LIN {X 0,Y 248.743,Z 466.9,A -85,B 0,C 180,E1 -20308.54,E2 -20308.54} C_VEL
LIN {X 0,Y 247.758,Z 471.99,A -85,B 0,C 180,E1 -20311.566,E2 -20311.566} C_VEL
LIN {X 0,Y 246.638,Z 476.028,A -85,B 0,C 180,E1 -20313.789,E2 -20313.789} C_VEL
LIN {X 0,Y 245.403,Z 479.129,A -85,B 0,C 180,E1 -20315.464,E2 -20315.464} C_VEL
LIN {X 0,Y 244.484,Z 480.76,A -85,B 0,C 180,E1 -20316.269,E2 -20316.269} C_VEL
LIN {X 0,Y 239.749,Z 485.852,A -85,B 0,C 180,E1 -20318.505,E2 -20318.505} C_VEL
LIN {X 0,Y 235.404,Z 489.582,A -85,B 0,C 180,E1 -20320.828,E2 -20320.828} C_VEL
LIN {X 0,Y 232.82,Z 491.419,A -85,B 0,C 180,E1 -20322.43,E2 -20322.43} C_VEL
LIN {X 0,Y 230.431,Z 492.703,A -85,B 0,C 180,E1 -20324.068,E2 -20324.068} C_VEL
LIN {X 0,Y 228.241,Z 493.449,A -85,B 0,C 180,E1 -20325.739,E2 -20325.739} C_VEL
LIN {X 0,Y 226.236,Z 493.719,A -85,B 0,C 180,E1 -20327.441,E2 -20327.441} C_VEL
LIN {X 0,Y 224.375,Z 493.441,A -85,B 0,C 180,E1 -20329.168,E2 -20329.168} C_VEL
LIN {X 0,Y 222.889,Z 492.598,A -85,B 0,C 180,E1 -20330.929,E2 -20330.929} C_VEL
LIN {X 0,Y 221.691,Z 491.23,A -85,B 0,C 180,E1 -20332.715,E2 -20332.715} C_VEL
LIN {X 0,Y 220.302,Z 488.075,A -85,B 0,C 180,E1 -20335.426,E2 -20335.426} C_VEL
LIN {X 0,Y 219.514,Z 483.587,A -85,B 0,C 180,E1 -20338.165,E2 -20338.165} C_VEL
LIN {X 0,Y 219.226,Z 477.6,A -85,B 0,C 180,E1 -20340.919,E2 -20340.919} C_VEL
LIN {X 0,Y 219.359,Z 471.25,A -85,B 0,C 180,E1 -20343.214,E2 -20343.214} C_VEL
LIN {X 0,Y 219.828,Z 463.432,A -85,B 0,C 180,E1 -20345.504,E2 -20345.504} C_VEL
LIN {X 0,Y 220.117,Z 454.301,A -85,B 0,C 180,E1 -20347.658,E2 -20347.658} C_VEL
LIN {X 0,Y 220.624,Z 443.788,A -85,B 0,C 180,E1 -20349.628,E2 -20349.628} C_VEL
LIN {X 0,Y 221.055,Z 434.685,A -85,B 0,C 180,E1 -20350.997,E2 -20350.997} C_VEL
LIN {X 0,Y 219.764,Z 422.117,A -85,B 0,C 180,E1 -20352.466,E2 -20352.466} C_VEL
LIN {X 0,Y 219.404,Z 416.978,A -85,B 0,C 180,E1 -20352.958,E2 -20352.958} C_VEL
LIN {X 0,Y 219.691,Z 410.88,A -85,B 0,C 180,E1 -20357.693,E2 -20357.693} C_VEL
LIN {X 0,Y 220.166,Z 404.789,A -85,B 0,C 180,E1 -20362.523,E2 -20362.523} C_VEL
LIN {X 0,Y 220.698,Z 399.342,A -85,B 0,C 180,E1 -20366.919,E2 -20366.919} C_VEL
LIN {X 0,Y 221.276,Z 394.44,A -85,B 0,C 180,E1 -20370.956,E2 -20370.956} C_VEL
LIN {X 0,Y 221.123,Z 392.931,A -85,B 0,C 180,E1 -20372.443,E2 -20372.443} C_VEL
LIN {X 0,Y 220.841,Z 392.976,A -85,B 0,C 180,E1 -20377.288,E2 -20377.288} C_VEL
LIN {X 0,Y 220.773,Z 392.981,A -85,B 0,C 180,E1 -20381.952,E2 -20381.952} C_VEL
LIN {X 0,Y 220.778,Z 392.982,A -85,B 0,C 180,E1 -20385.547,E2 -20385.547} C_VEL
LIN {X 0,Y 220.809,Z 392.979,A -85,B 0,C 180,E1 -20390.463,E2 -20390.463} C_VEL
LIN {X 0,Y 220.803,Z 392.98,A -85,B 0,C 180,E1 -20395.045,E2 -20395.045} C_VEL
LIN {X 0,Y 220.871,Z 392.968,A -85,B 0,C 180,E1 -20399.395,E2 -20399.395} C_VEL
LIN {X 0,Y 220.898,Z 392.967,A -85,B 0,C 180,E1 -20403.55,E2 -20403.55} C_VEL
LIN {X 0,Y 220.882,Z 392.967,A -85,B 0,C 180,E1 -20407.554,E2 -20407.554} C_VEL
LIN {X 0,Y 220.988,Z 392.958,A -85,B 0,C 180,E1 -20412.571,E2 -20412.571} C_VEL
LIN {X 0,Y 221.015,Z 392.949,A -85,B 0,C 180,E1 -20417.139,E2 -20417.139} C_VEL
LIN {X 0,Y 221.208,Z 392.929,A -85,B 0,C 180,E1 -20420.859,E2 -20420.859} C_VEL
LIN {X 0,Y 221.263,Z 392.922,A -85,B 0,C 180,E1 -20422.701,E2 -20422.701} C_VEL
LIN {X 0,Y 221.515,Z 392.893,A -85,B 0,C 180,E1 -20428.182,E2 -20428.182} C_VEL
LIN {X 0,Y 221.516,Z 392.893,A -85,B 0,C 180,E1 -20431.818,E2 -20431.818} C_VEL
LIN {X 0,Y 221.292,Z 392.918,A -85,B 0,C 180,E1 -20437.298,E2 -20437.298} C_VEL
LIN {X 0,Y 221.115,Z 392.939,A -85,B 0,C 180,E1 -20440.994,E2 -20440.994} C_VEL
LIN {X 0,Y 221.02,Z 392.952,A -85,B 0,C 180,E1 -20446.629,E2 -20446.629} C_VEL
LIN {X 0,Y 220.913,Z 392.963,A -85,B 0,C 180,E1 -20450.484,E2 -20450.484} C_VEL
LIN {X 0,Y 220.875,Z 392.97,A -85,B 0,C 180,E1 -20454.434,E2 -20454.434} C_VEL
LIN {X 0,Y 220.838,Z 392.973,A -85,B 0,C 180,E1 -20458.513,E2 -20458.513} C_VEL
LIN {X 0,Y 220.827,Z 392.976,A -85,B 0,C 180,E1 -20462.754,E2 -20462.754} C_VEL
LIN {X 0,Y 220.84,Z 392.976,A -85,B 0,C 180,E1 -20467.288,E2 -20467.288} C_VEL
LIN {X 0,Y 220.773,Z 392.983,A -85,B 0,C 180,E1 -20471.952,E2 -20471.952} C_VEL
LIN {X 0,Y 220.769,Z 392.983,A -85,B 0,C 180,E1 -20475.544,E2 -20475.544} C_VEL
LIN {X 0,Y 220.808,Z 392.978,A -85,B 0,C 180,E1 -20480.463,E2 -20480.463} C_VEL
LIN {X 0,Y 220.802,Z 392.979,A -85,B 0,C 180,E1 -20485.045,E2 -20485.045} C_VEL
LIN {X 0,Y 220.87,Z 392.972,A -85,B 0,C 180,E1 -20489.395,E2 -20489.395} C_VEL
LIN {X 0,Y 220.897,Z 392.965,A -85,B 0,C 180,E1 -20493.549,E2 -20493.549} C_VEL
LIN {X 0,Y 220.88,Z 392.97,A -85,B 0,C 180,E1 -20497.553,E2 -20497.553} C_VEL
LIN {X 0,Y 220.986,Z 392.956,A -85,B 0,C 180,E1 -20502.571,E2 -20502.571} C_VEL
LIN {X 0,Y 221.029,Z 392.952,A -85,B 0,C 180,E1 -20507.139,E2 -20507.139} C_VEL
LIN {X 0,Y 221.26,Z 392.921,A -85,B 0,C 180,E1 -20510.862,E2 -20510.862} C_VEL
LIN {X 0,Y 221.313,Z 392.917,A -85,B 0,C 180,E1 -20512.702,E2 -20512.702} C_VEL
LIN {X 0,Y 221.515,Z 392.891,A -85,B 0,C 180,E1 -20518.182,E2 -20518.182} C_VEL
LIN {X 0,Y 221.517,Z 392.889,A -85,B 0,C 180,E1 -20521.818,E2 -20521.818} C_VEL
LIN {X 0,Y 221.313,Z 392.913,A -85,B 0,C 180,E1 -20527.298,E2 -20527.298} C_VEL
LIN {X 0,Y 221.119,Z 392.94,A -85,B 0,C 180,E1 -20530.994,E2 -20530.994} C_VEL
LIN {X 0,Y 221.018,Z 392.95,A -85,B 0,C 180,E1 -20536.63,E2 -20536.63} C_VEL
LIN {X 0,Y 220.894,Z 392.969,A -85,B 0,C 180,E1 -20540.486,E2 -20540.486} C_VEL
LIN {X 0,Y 220.869,Z 392.97,A -85,B 0,C 180,E1 -20544.435,E2 -20544.435} C_VEL
LIN {X 0,Y 220.828,Z 392.977,A -85,B 0,C 180,E1 -20548.515,E2 -20548.515} C_VEL
LIN {X 0,Y 220.824,Z 392.975,A -85,B 0,C 180,E1 -20552.755,E2 -20552.755} C_VEL
LIN {X 0,Y 220.839,Z 392.975,A -85,B 0,C 180,E1 -20557.288,E2 -20557.288} C_VEL
LIN {X 0,Y 220.777,Z 392.981,A -85,B 0,C 180,E1 -20561.951,E2 -20561.951} C_VEL
LIN {X 0,Y 220.889,Z 392.973,A -85,B 0,C 180,E1 -20565.812,E2 -20565.812} C_VEL
LIN {X 0,Y 222.459,Z 401.177,A -85,B 0,C 180,E1 -20570.814,E2 -20570.814} C_VEL
LIN {X 0,Y 223.883,Z 407.84,A -85,B 0,C 180,E1 -20574.704,E2 -20574.704} C_VEL
LIN {X 0,Y 225.236,Z 413.607,A -85,B 0,C 180,E1 -20577.964,E2 -20577.964} C_VEL
LIN {X 0,Y 225.146,Z 415.498,A -85,B 0,C 180,E1 -20578.999,E2 -20578.999} C_VEL
LIN {X 0,Y 222.346,Z 426.144,A -85,B 0,C 180,E1 -20584.741,E2 -20584.741} C_VEL
LIN {X 0,Y 220.633,Z 436.118,A -85,B 0,C 180,E1 -20590.218,E2 -20590.218} C_VEL
LIN {X 0,Y 220.815,Z 450.1,A -85,B 0,C 180,E1 -20591.321,E2 -20591.321} C_VEL
LIN {X 0,Y 221.565,Z 462.255,A -85,B 0,C 180,E1 -20592.619,E2 -20592.619} C_VEL
LIN {X 0,Y 221.177,Z 467.503,A -85,B 0,C 180,E1 -20593.309,E2 -20593.309} C_VEL
LIN {X 0,Y 219.653,Z 472.431,A -85,B 0,C 180,E1 -20594.084,E2 -20594.084} C_VEL
LIN {X 0,Y 215.142,Z 483.065,A -85,B 0,C 180,E1 -20596.213,E2 -20596.213} C_VEL
LIN {X 0,Y 214.264,Z 487.568,A -85,B 0,C 180,E1 -20597.255,E2 -20597.255} C_VEL
LIN {X 0,Y 213.864,Z 496.597,A -85,B 0,C 180,E1 -20599.588,E2 -20599.588} C_VEL
LIN {X 0,Y 213.658,Z 503.978,A -85,B 0,C 180,E1 -20601.94,E2 -20601.94} C_VEL
LIN {X 0,Y 213.802,Z 510.152,A -85,B 0,C 180,E1 -20604.341,E2 -20604.341} C_VEL
LIN {X 0,Y 213.841,Z 515.818,A -85,B 0,C 180,E1 -20607.174,E2 -20607.174} C_VEL
LIN {X 0,Y 213.76,Z 518.769,A -85,B 0,C 180,E1 -20609.058,E2 -20609.058} C_VEL
LIN {X 0,Y 213.37,Z 522.06,A -85,B 0,C 180,E1 -20611.888,E2 -20611.888} C_VEL
LIN {X 0,Y 212.82,Z 523.57,A -85,B 0,C 180,E1 -20613.787,E2 -20613.787} C_VEL
LIN {X 0,Y 212.266,Z 525.354,A -85,B 0,C 180,E1 -20617.611,E2 -20617.611} C_VEL
LIN {X 0,Y 212.516,Z 525.684,A -85,B 0,C 180,E1 -20621.445,E2 -20621.445} C_VEL
LIN {X 0,Y 213.939,Z 524.599,A -85,B 0,C 180,E1 -20625.237,E2 -20625.237} C_VEL
LIN {X 0,Y 216.51,Z 522.127,A -85,B 0,C 180,E1 -20628.942,E2 -20628.942} C_VEL
LIN {X 0,Y 220.264,Z 518.23,A -85,B 0,C 180,E1 -20632.513,E2 -20632.513} C_VEL
LIN {X 0,Y 223.867,Z 514.286,A -85,B 0,C 180,E1 -20635.076,E2 -20635.076} C_VEL
LIN {X 0,Y 229.577,Z 507.575,A -85,B 0,C 180,E1 -20638.327,E2 -20638.327} C_VEL
LIN {X 0,Y 234.674,Z 501.249,A -85,B 0,C 180,E1 -20640.605,E2 -20640.605} C_VEL
LIN {X 0,Y 239.782,Z 493.834,A -85,B 0,C 180,E1 -20642.836,E2 -20642.836} C_VEL
LIN {X 0,Y 243.085,Z 487.19,A -85,B 0,C 180,E1 -20644.821,E2 -20644.821} C_VEL
LIN {X 0,Y 246.585,Z 477.943,A -85,B 0,C 180,E1 -20647.627,E2 -20647.627} C_VEL
LIN {X 0,Y 247.275,Z 475.617,A -85,B 0,C 180,E1 -20648.373,E2 -20648.373} C_VEL
LIN {X 0,Y 247.04,Z 473.044,A -85,B 0,C 180,E1 -20649.815,E2 -20649.815} C_VEL
LIN {X 0,Y 246.243,Z 470.086,A -85,B 0,C 180,E1 -20652.092,E2 -20652.092} C_VEL
LIN {X 0,Y 245.716,Z 467.717,A -85,B 0,C 180,E1 -20654.352,E2 -20654.352} C_VEL
LIN {X 0,Y 245.265,Z 466.253,A -85,B 0,C 180,E1 -20656.551,E2 -20656.551} C_VEL
LIN {X 0,Y 244.953,Z 465.624,A -85,B 0,C 180,E1 -20658.708,E2 -20658.708} C_VEL
LIN {X 0,Y 244.685,Z 465.81,A -85,B 0,C 180,E1 -20660.852,E2 -20660.852} C_VEL
LIN {X 0,Y 244.47,Z 466.992,A -85,B 0,C 180,E1 -20663.605,E2 -20663.605} C_VEL
LIN {X 0,Y 244.352,Z 467.904,A -85,B 0,C 180,E1 -20664.884,E2 -20664.884} C_VEL
LIN {X 0,Y 244.034,Z 469.82,A -85,B 0,C 180,E1 -20666.826,E2 -20666.826} C_VEL
LIN {X 0,Y 243.396,Z 472.34,A -85,B 0,C 180,E1 -20668.685,E2 -20668.685} C_VEL
LIN {X 0,Y 242.066,Z 476.535,A -85,B 0,C 180,E1 -20671.432,E2 -20671.432} C_VEL
LIN {X 0,Y 240.286,Z 480.703,A -85,B 0,C 180,E1 -20673.977,E2 -20673.977} C_VEL
LIN {X 0,Y 239.559,Z 482.111,A -85,B 0,C 180,E1 -20674.825,E2 -20674.825} C_VEL
LIN {X 0,Y 238.383,Z 483.655,A -85,B 0,C 180,E1 -20675.622,E2 -20675.622} C_VEL
LIN {X 0,Y 233.427,Z 488.207,A -85,B 0,C 180,E1 -20677.892,E2 -20677.892} C_VEL
LIN {X 0,Y 228.932,Z 491.524,A -85,B 0,C 180,E1 -20680.264,E2 -20680.264} C_VEL
LIN {X 0,Y 226.222,Z 493.059,A -85,B 0,C 180,E1 -20681.901,E2 -20681.901} C_VEL
LIN {X 0,Y 223.744,Z 494.077,A -85,B 0,C 180,E1 -20683.579,E2 -20683.579} C_VEL
LIN {X 0,Y 221.453,Z 494.605,A -85,B 0,C 180,E1 -20685.292,E2 -20685.292} C_VEL
LIN {X 0,Y 219.356,Z 494.613,A -85,B 0,C 180,E1 -20687.04,E2 -20687.04} C_VEL
LIN {X 0,Y 217.444,Z 494.086,A -85,B 0,C 180,E1 -20688.818,E2 -20688.818} C_VEL
LIN {X 0,Y 215.906,Z 493.026,A -85,B 0,C 180,E1 -20690.633,E2 -20690.633} C_VEL
LIN {X 0,Y 214.127,Z 490.391,A -85,B 0,C 180,E1 -20693.404,E2 -20693.404} C_VEL
LIN {X 0,Y 212.882,Z 486.483,A -85,B 0,C 180,E1 -20696.214,E2 -20696.214} C_VEL
LIN {X 0,Y 212.297,Z 481.155,A -85,B 0,C 180,E1 -20699.052,E2 -20699.052} C_VEL
LIN {X 0,Y 212.165,Z 474.239,A -85,B 0,C 180,E1 -20701.898,E2 -20701.898} C_VEL
LIN {X 0,Y 212.495,Z 466.979,A -85,B 0,C 180,E1 -20704.268,E2 -20704.268} C_VEL
LIN {X 0,Y 212.873,Z 459.912,A -85,B 0,C 180,E1 -20706.16,E2 -20706.16} C_VEL
LIN {X 0,Y 213.245,Z 450.42,A -85,B 0,C 180,E1 -20708.251,E2 -20708.251} C_VEL
LIN {X 0,Y 213.741,Z 439.494,A -85,B 0,C 180,E1 -20710.18,E2 -20710.18} C_VEL
LIN {X 0,Y 213.97,Z 434.77,A -85,B 0,C 180,E1 -20710.887,E2 -20710.887} C_VEL
LIN {X 0,Y 212.789,Z 423.368,A -85,B 0,C 180,E1 -20712.276,E2 -20712.276} C_VEL
LIN {X 0,Y 212.331,Z 417.259,A -85,B 0,C 180,E1 -20712.91,E2 -20712.91} C_VEL
LIN {X 0,Y 212.669,Z 410.519,A -85,B 0,C 180,E1 -20718.297,E2 -20718.297} C_VEL
LIN {X 0,Y 213.197,Z 404.385,A -85,B 0,C 180,E1 -20723.302,E2 -20723.302} C_VEL
LIN {X 0,Y 213.882,Z 398.208,A -85,B 0,C 180,E1 -20728.455,E2 -20728.455} C_VEL
LIN {X 0,Y 214.245,Z 394.452,A -85,B 0,C 180,E1 -20731.659,E2 -20731.659} C_VEL
LIN {X 0,Y 214.104,Z 393.807,A -85,B 0,C 180,E1 -20732.236,E2 -20732.236} C_VEL
LIN {X 0,Y 213.754,Z 393.857,A -85,B 0,C 180,E1 -20737.898,E2 -20737.898} C_VEL
LIN {X 0,Y 213.715,Z 393.861,A -85,B 0,C 180,E1 -20741.125,E2 -20741.125} C_VEL
LIN {X 0,Y 213.71,Z 393.86,A -85,B 0,C 180,E1 -20743.678,E2 -20743.678} C_VEL
LIN {X 0,Y 213.71,Z 393.864,A -85,B 0,C 180,E1 -20746.343,E2 -20746.343} C_VEL
LIN {X 0,Y 213.72,Z 393.861,A -85,B 0,C 180,E1 -20749.143,E2 -20749.143} C_VEL
LIN {X 0,Y 213.746,Z 393.857,A -85,B 0,C 180,E1 -20753.712,E2 -20753.712} C_VEL
LIN {X 0,Y 213.77,Z 393.856,A -85,B 0,C 180,E1 -20758.263,E2 -20758.263} C_VEL
LIN {X 0,Y 213.829,Z 393.85,A -85,B 0,C 180,E1 -20762.603,E2 -20762.603} C_VEL
LIN {X 0,Y 213.855,Z 393.843,A -85,B 0,C 180,E1 -20766.953,E2 -20766.953} C_VEL
LIN {X 0,Y 213.936,Z 393.838,A -85,B 0,C 180,E1 -20772.305,E2 -20772.305} C_VEL
LIN {X 0,Y 213.956,Z 393.829,A -85,B 0,C 180,E1 -20776.707,E2 -20776.707} C_VEL
LIN {X 0,Y 214.145,Z 393.81,A -85,B 0,C 180,E1 -20780.555,E2 -20780.555} C_VEL
LIN {X 0,Y 214.104,Z 393.813,A -85,B 0,C 180,E1 -20784.348,E2 -20784.348} C_VEL
LIN {X 0,Y 214.449,Z 393.773,A -85,B 0,C 180,E1 -20788.122,E2 -20788.122} C_VEL
LIN {X 0,Y 214.553,Z 393.761,A -85,B 0,C 180,E1 -20790,E2 -20790} C_VEL
LIN {X 0,Y 214.45,Z 393.773,A -85,B 0,C 180,E1 -20791.878,E2 -20791.878} C_VEL
LIN {X 0,Y 214.23,Z 393.799,A -85,B 0,C 180,E1 -20797.54,E2 -20797.54} C_VEL
LIN {X 0,Y 214.048,Z 393.821,A -85,B 0,C 180,E1 -20801.362,E2 -20801.362} C_VEL
LIN {X 0,Y 213.937,Z 393.834,A -85,B 0,C 180,E1 -20805.237,E2 -20805.237} C_VEL
LIN {X 0,Y 213.879,Z 393.842,A -85,B 0,C 180,E1 -20809.184,E2 -20809.184} C_VEL
LIN {X 0,Y 213.858,Z 393.843,A -85,B 0,C 180,E1 -20813.226,E2 -20813.226} C_VEL
LIN {X 0,Y 213.831,Z 393.85,A -85,B 0,C 180,E1 -20817.45,E2 -20817.45} C_VEL
LIN {X 0,Y 213.782,Z 393.855,A -85,B 0,C 180,E1 -20821.735,E2 -20821.735} C_VEL
LIN {X 0,Y 213.755,Z 393.856,A -85,B 0,C 180,E1 -20826.286,E2 -20826.286} C_VEL
LIN {X 0,Y 213.716,Z 393.863,A -85,B 0,C 180,E1 -20831.124,E2 -20831.124} C_VEL
LIN {X 0,Y 213.704,Z 393.864,A -85,B 0,C 180,E1 -20833.679,E2 -20833.679} C_VEL
LIN {X 0,Y 213.704,Z 393.861,A -85,B 0,C 180,E1 -20836.345,E2 -20836.345} C_VEL
LIN {X 0,Y 213.718,Z 393.863,A -85,B 0,C 180,E1 -20839.143,E2 -20839.143} C_VEL
LIN {X 0,Y 213.745,Z 393.857,A -85,B 0,C 180,E1 -20843.712,E2 -20843.712} C_VEL
LIN {X 0,Y 213.797,Z 393.853,A -85,B 0,C 180,E1 -20848.725,E2 -20848.725} C_VEL
LIN {X 0,Y 213.827,Z 393.849,A -85,B 0,C 180,E1 -20852.603,E2 -20852.603} C_VEL
LIN {X 0,Y 213.854,Z 393.848,A -85,B 0,C 180,E1 -20856.953,E2 -20856.953} C_VEL
LIN {X 0,Y 213.934,Z 393.833,A -85,B 0,C 180,E1 -20862.305,E2 -20862.305} C_VEL
LIN {X 0,Y 213.983,Z 393.832,A -85,B 0,C 180,E1 -20866.708,E2 -20866.708} C_VEL
LIN {X 0,Y 214.199,Z 393.802,A -85,B 0,C 180,E1 -20870.558,E2 -20870.558} C_VEL
LIN {X 0,Y 214.25,Z 393.794,A -85,B 0,C 180,E1 -20872.46,E2 -20872.46} C_VEL
LIN {X 0,Y 214.448,Z 393.771,A -85,B 0,C 180,E1 -20878.122,E2 -20878.122} C_VEL
LIN {X 0,Y 214.553,Z 393.755,A -85,B 0,C 180,E1 -20880,E2 -20880} C_VEL
LIN {X 0,Y 214.45,Z 393.769,A -85,B 0,C 180,E1 -20881.878,E2 -20881.878} C_VEL
LIN {X 0,Y 214.25,Z 393.793,A -85,B 0,C 180,E1 -20887.539,E2 -20887.539} C_VEL
LIN {X 0,Y 214.049,Z 393.82,A -85,B 0,C 180,E1 -20891.362,E2 -20891.362} C_VEL
LIN {X 0,Y 213.935,Z 393.833,A -85,B 0,C 180,E1 -20895.237,E2 -20895.237} C_VEL
LIN {X 0,Y 213.841,Z 393.845,A -85,B 0,C 180,E1 -20899.187,E2 -20899.187} C_VEL
LIN {X 0,Y 213.849,Z 393.845,A -85,B 0,C 180,E1 -20903.227,E2 -20903.227} C_VEL
LIN {X 0,Y 213.83,Z 393.846,A -85,B 0,C 180,E1 -20907.45,E2 -20907.45} C_VEL
LIN {X 0,Y 213.771,Z 393.857,A -85,B 0,C 180,E1 -20911.737,E2 -20911.737} C_VEL
LIN {X 0,Y 213.754,Z 393.858,A -85,B 0,C 180,E1 -20916.286,E2 -20916.286} C_VEL
LIN {X 0,Y 213.718,Z 393.861,A -85,B 0,C 180,E1 -20921.124,E2 -20921.124} C_VEL
LIN {X 0,Y 213.845,Z 393.927,A -85,B 0,C 180,E1 -20925.628,E2 -20925.628} C_VEL
LIN {X 0,Y 215.277,Z 401.464,A -85,B 0,C 180,E1 -20930.397,E2 -20930.397} C_VEL
LIN {X 0,Y 216.886,Z 408.878,A -85,B 0,C 180,E1 -20934.888,E2 -20934.888} C_VEL
LIN {X 0,Y 218.154,Z 414.264,A -85,B 0,C 180,E1 -20938.047,E2 -20938.047} C_VEL
LIN {X 0,Y 218.011,Z 415.857,A -85,B 0,C 180,E1 -20938.95,E2 -20938.95} C_VEL
LIN {X 0,Y 215.155,Z 426.4,A -85,B 0,C 180,E1 -20944.872,E2 -20944.872} C_VEL
LIN {X 0,Y 213.561,Z 435.845,A -85,B 0,C 180,E1 -20950.287,E2 -20950.287} C_VEL
LIN {X 0,Y 213.676,Z 448.936,A -85,B 0,C 180,E1 -20951.344,E2 -20951.344} C_VEL
LIN {X 0,Y 214.525,Z 462.513,A -85,B 0,C 180,E1 -20952.852,E2 -20952.852} C_VEL
LIN {X 0,Y 215.247,Z 471.51,A -85,B 0,C 180,E1 -20954.13,E2 -20954.13} C_VEL
LIN {X 0,Y 214.623,Z 481.89,A -85,B 0,C 180,E1 -20956.025,E2 -20956.025} C_VEL
LIN {X 0,Y 214.264,Z 487.568,A -85,B 0,C 180,E1 -20957.255,E2 -20957.255} C_VEL
LIN {X 0,Y 213.411,Z 491.817,A -85,B 0,C 180,E1 -20958.335,E2 -20958.335} C_VEL
LIN {X 0,Y 210.34,Z 497.938,A -85,B 0,C 180,E1 -20960.277,E2 -20960.277} C_VEL
LIN {X 0,Y 207.438,Z 503.473,A -85,B 0,C 180,E1 -20962.415,E2 -20962.415} C_VEL
LIN {X 0,Y 206.869,Z 506.757,A -85,B 0,C 180,E1 -20963.78,E2 -20963.78} C_VEL
LIN {X 0,Y 206.918,Z 511.845,A -85,B 0,C 180,E1 -20966.105,E2 -20966.105} C_VEL
LIN {X 0,Y 206.926,Z 516.83,A -85,B 0,C 180,E1 -20969.027,E2 -20969.027} C_VEL
LIN {X 0,Y 206.469,Z 520.34,A -85,B 0,C 180,E1 -20971.951,E2 -20971.951} C_VEL
LIN {X 0,Y 205.508,Z 523.233,A -85,B 0,C 180,E1 -20975.889,E2 -20975.889} C_VEL
LIN {X 0,Y 205.324,Z 524.57,A -85,B 0,C 180,E1 -20979.855,E2 -20979.855} C_VEL
LIN {X 0,Y 206.105,Z 524.49,A -85,B 0,C 180,E1 -20983.81,E2 -20983.81} C_VEL
LIN {X 0,Y 208.268,Z 523.06,A -85,B 0,C 180,E1 -20987.68,E2 -20987.68} C_VEL
LIN {X 0,Y 211.572,Z 520.267,A -85,B 0,C 180,E1 -20991.432,E2 -20991.432} C_VEL
LIN {X 0,Y 216.125,Z 516.029,A -85,B 0,C 180,E1 -20995.008,E2 -20995.008} C_VEL
LIN {X 0,Y 221.832,Z 510.272,A -85,B 0,C 180,E1 -20998.374,E2 -20998.374} C_VEL
LIN {X 0,Y 228.7,Z 502.714,A -85,B 0,C 180,E1 -21001.495,E2 -21001.495} C_VEL
LIN {X 0,Y 234.074,Z 495.802,A -85,B 0,C 180,E1 -21003.743,E2 -21003.743} C_VEL
LIN {X 0,Y 237.657,Z 489.653,A -85,B 0,C 180,E1 -21005.736,E2 -21005.736} C_VEL
LIN {X 0,Y 241.689,Z 480.782,A -85,B 0,C 180,E1 -21008.645,E2 -21008.645} C_VEL
LIN {X 0,Y 242.148,Z 479.508,A -85,B 0,C 180,E1 -21009.118,E2 -21009.118} C_VEL
LIN {X 0,Y 241.82,Z 476.811,A -85,B 0,C 180,E1 -21010.919,E2 -21010.919} C_VEL
LIN {X 0,Y 241.097,Z 473.14,A -85,B 0,C 180,E1 -21014.395,E2 -21014.395} C_VEL
LIN {X 0,Y 240.662,Z 471.59,A -85,B 0,C 180,E1 -21016.893,E2 -21016.893} C_VEL
LIN {X 0,Y 240.138,Z 471.113,A -85,B 0,C 180,E1 -21019.92,E2 -21019.92} C_VEL
LIN {X 0,Y 239.779,Z 471.659,A -85,B 0,C 180,E1 -21022.315,E2 -21022.315} C_VEL
LIN {X 0,Y 239.515,Z 472.537,A -85,B 0,C 180,E1 -21024.066,E2 -21024.066} C_VEL
LIN {X 0,Y 239.055,Z 474.137,A -85,B 0,C 180,E1 -21026.042,E2 -21026.042} C_VEL
LIN {X 0,Y 238.25,Z 476.24,A -85,B 0,C 180,E1 -21027.929,E2 -21027.929} C_VEL
LIN {X 0,Y 236.606,Z 479.884,A -85,B 0,C 180,E1 -21030.653,E2 -21030.653} C_VEL
LIN {X 0,Y 234.5,Z 483.698,A -85,B 0,C 180,E1 -21033.285,E2 -21033.285} C_VEL
LIN {X 0,Y 233.681,Z 484.944,A -85,B 0,C 180,E1 -21034.145,E2 -21034.145} C_VEL
LIN {X 0,Y 232.279,Z 486.419,A -85,B 0,C 180,E1 -21034.938,E2 -21034.938} C_VEL
LIN {X 0,Y 227.131,Z 490.472,A -85,B 0,C 180,E1 -21037.246,E2 -21037.246} C_VEL
LIN {X 0,Y 222.456,Z 493.355,A -85,B 0,C 180,E1 -21039.664,E2 -21039.664} C_VEL
LIN {X 0,Y 219.631,Z 494.616,A -85,B 0,C 180,E1 -21041.338,E2 -21041.338} C_VEL
LIN {X 0,Y 217.044,Z 495.367,A -85,B 0,C 180,E1 -21043.057,E2 -21043.057} C_VEL
LIN {X 0,Y 214.674,Z 495.645,A -85,B 0,C 180,E1 -21044.817,E2 -21044.817} C_VEL
LIN {X 0,Y 212.475,Z 495.394,A -85,B 0,C 180,E1 -21046.612,E2 -21046.612} C_VEL
LIN {X 0,Y 210.524,Z 494.633,A -85,B 0,C 180,E1 -21048.446,E2 -21048.446} C_VEL
LIN {X 0,Y 208.931,Z 493.335,A -85,B 0,C 180,E1 -21050.318,E2 -21050.318} C_VEL
LIN {X 0,Y 207.072,Z 490.342,A -85,B 0,C 180,E1 -21053.178,E2 -21053.178} C_VEL
LIN {X 0,Y 205.806,Z 486.094,A -85,B 0,C 180,E1 -21056.084,E2 -21056.084} C_VEL
LIN {X 0,Y 205.219,Z 480.408,A -85,B 0,C 180,E1 -21059.019,E2 -21059.019} C_VEL
LIN {X 0,Y 205.148,Z 473.053,A -85,B 0,C 180,E1 -21061.963,E2 -21061.963} C_VEL
LIN {X 0,Y 205.634,Z 463.716,A -85,B 0,C 180,E1 -21064.902,E2 -21064.902} C_VEL
LIN {X 0,Y 205.903,Z 454.829,A -85,B 0,C 180,E1 -21067.108,E2 -21067.108} C_VEL
LIN {X 0,Y 206.455,Z 443.767,A -85,B 0,C 180,E1 -21069.296,E2 -21069.296} C_VEL
LIN {X 0,Y 206.86,Z 434.513,A -85,B 0,C 180,E1 -21070.77,E2 -21070.77} C_VEL
LIN {X 0,Y 205.629,Z 422.859,A -85,B 0,C 180,E1 -21072.209,E2 -21072.209} C_VEL
LIN {X 0,Y 205.263,Z 417.59,A -85,B 0,C 180,E1 -21072.796,E2 -21072.796} C_VEL
LIN {X 0,Y 205.55,Z 411.351,A -85,B 0,C 180,E1 -21077.922,E2 -21077.922} C_VEL
LIN {X 0,Y 206.073,Z 405.346,A -85,B 0,C 180,E1 -21082.953,E2 -21082.953} C_VEL
LIN {X 0,Y 206.792,Z 398.969,A -85,B 0,C 180,E1 -21088.412,E2 -21088.412} C_VEL
LIN {X 0,Y 207.122,Z 396.445,A -85,B 0,C 180,E1 -21090.596,E2 -21090.596} C_VEL
LIN {X 0,Y 207.051,Z 394.684,A -85,B 0,C 180,E1 -21092.356,E2 -21092.356} C_VEL
LIN {X 0,Y 206.704,Z 394.735,A -85,B 0,C 180,E1 -21097.735,E2 -21097.735} C_VEL
LIN {X 0,Y 206.645,Z 394.74,A -85,B 0,C 180,E1 -21101.563,E2 -21101.563} C_VEL
LIN {X 0,Y 206.637,Z 394.743,A -85,B 0,C 180,E1 -21105.581,E2 -21105.581} C_VEL
LIN {X 0,Y 206.663,Z 394.739,A -85,B 0,C 180,E1 -21109.749,E2 -21109.749} C_VEL
LIN {X 0,Y 206.701,Z 394.739,A -85,B 0,C 180,E1 -21114.689,E2 -21114.689} C_VEL
LIN {X 0,Y 206.716,Z 394.73,A -85,B 0,C 180,E1 -21119.338,E2 -21119.338} C_VEL
LIN {X 0,Y 206.736,Z 394.732,A -85,B 0,C 180,E1 -21123.772,E2 -21123.772} C_VEL
LIN {X 0,Y 206.761,Z 394.728,A -85,B 0,C 180,E1 -21128.043,E2 -21128.043} C_VEL
LIN {X 0,Y 206.88,Z 394.716,A -85,B 0,C 180,E1 -21132.197,E2 -21132.197} C_VEL
LIN {X 0,Y 206.899,Z 394.71,A -85,B 0,C 180,E1 -21136.244,E2 -21136.244} C_VEL
LIN {X 0,Y 207.102,Z 394.689,A -85,B 0,C 180,E1 -21140.231,E2 -21140.231} C_VEL
LIN {X 0,Y 207.065,Z 394.691,A -85,B 0,C 180,E1 -21144.156,E2 -21144.156} C_VEL
LIN {X 0,Y 207.385,Z 394.652,A -85,B 0,C 180,E1 -21148.058,E2 -21148.058} C_VEL
LIN {X 0,Y 207.518,Z 394.637,A -85,B 0,C 180,E1 -21150,E2 -21150} C_VEL
LIN {X 0,Y 207.386,Z 394.652,A -85,B 0,C 180,E1 -21151.942,E2 -21151.942} C_VEL
LIN {X 0,Y 207.17,Z 394.68,A -85,B 0,C 180,E1 -21157.799,E2 -21157.799} C_VEL
LIN {X 0,Y 206.985,Z 394.7,A -85,B 0,C 180,E1 -21161.755,E2 -21161.755} C_VEL
LIN {X 0,Y 206.871,Z 394.717,A -85,B 0,C 180,E1 -21165.77,E2 -21165.77} C_VEL
LIN {X 0,Y 206.816,Z 394.721,A -85,B 0,C 180,E1 -21169.866,E2 -21169.866} C_VEL
LIN {X 0,Y 206.771,Z 394.728,A -85,B 0,C 180,E1 -21174.071,E2 -21174.071} C_VEL
LIN {X 0,Y 206.746,Z 394.728,A -85,B 0,C 180,E1 -21178.418,E2 -21178.418} C_VEL
LIN {X 0,Y 206.711,Z 394.735,A -85,B 0,C 180,E1 -21182.955,E2 -21182.955} C_VEL
LIN {X 0,Y 206.724,Z 394.736,A -85,B 0,C 180,E1 -21185.32,E2 -21185.32} C_VEL
LIN {X 0,Y 206.667,Z 394.738,A -85,B 0,C 180,E1 -21190.25,E2 -21190.25} C_VEL
LIN {X 0,Y 206.632,Z 394.743,A -85,B 0,C 180,E1 -21195.582,E2 -21195.582} C_VEL
LIN {X 0,Y 206.661,Z 394.741,A -85,B 0,C 180,E1 -21199.748,E2 -21199.748} C_VEL
LIN {X 0,Y 206.7,Z 394.735,A -85,B 0,C 180,E1 -21204.689,E2 -21204.689} C_VEL
LIN {X 0,Y 206.725,Z 394.734,A -85,B 0,C 180,E1 -21209.339,E2 -21209.339} C_VEL
LIN {X 0,Y 206.734,Z 394.728,A -85,B 0,C 180,E1 -21213.772,E2 -21213.772} C_VEL
LIN {X 0,Y 206.76,Z 394.728,A -85,B 0,C 180,E1 -21218.043,E2 -21218.043} C_VEL
LIN {X 0,Y 206.878,Z 394.712,A -85,B 0,C 180,E1 -21222.197,E2 -21222.197} C_VEL
LIN {X 0,Y 206.916,Z 394.709,A -85,B 0,C 180,E1 -21226.246,E2 -21226.246} C_VEL
LIN {X 0,Y 207.135,Z 394.681,A -85,B 0,C 180,E1 -21230.232,E2 -21230.232} C_VEL
LIN {X 0,Y 207.191,Z 394.672,A -85,B 0,C 180,E1 -21232.202,E2 -21232.202} C_VEL
LIN {X 0,Y 207.385,Z 394.651,A -85,B 0,C 180,E1 -21238.058,E2 -21238.058} C_VEL
LIN {X 0,Y 207.517,Z 394.632,A -85,B 0,C 180,E1 -21240,E2 -21240} C_VEL
LIN {X 0,Y 207.387,Z 394.649,A -85,B 0,C 180,E1 -21241.942,E2 -21241.942} C_VEL
LIN {X 0,Y 207.191,Z 394.673,A -85,B 0,C 180,E1 -21247.798,E2 -21247.798} C_VEL
LIN {X 0,Y 206.985,Z 394.701,A -85,B 0,C 180,E1 -21251.755,E2 -21251.755} C_VEL
LIN {X 0,Y 206.869,Z 394.715,A -85,B 0,C 180,E1 -21255.77,E2 -21255.77} C_VEL
LIN {X 0,Y 206.785,Z 394.726,A -85,B 0,C 180,E1 -21259.869,E2 -21259.869} C_VEL
LIN {X 0,Y 206.765,Z 394.729,A -85,B 0,C 180,E1 -21264.072,E2 -21264.072} C_VEL
LIN {X 0,Y 206.738,Z 394.732,A -85,B 0,C 180,E1 -21268.42,E2 -21268.42} C_VEL
LIN {X 0,Y 206.707,Z 394.733,A -85,B 0,C 180,E1 -21272.956,E2 -21272.956} C_VEL
LIN {X 0,Y 206.723,Z 394.73,A -85,B 0,C 180,E1 -21275.32,E2 -21275.32} C_VEL
LIN {X 0,Y 206.668,Z 394.74,A -85,B 0,C 180,E1 -21280.25,E2 -21280.25} C_VEL
LIN {X 0,Y 206.798,Z 394.734,A -85,B 0,C 180,E1 -21285.374,E2 -21285.374} C_VEL
LIN {X 0,Y 208.158,Z 401.926,A -85,B 0,C 180,E1 -21290.097,E2 -21290.097} C_VEL
LIN {X 0,Y 209.672,Z 408.914,A -85,B 0,C 180,E1 -21294.496,E2 -21294.496} C_VEL
LIN {X 0,Y 210.976,Z 414.306,A -85,B 0,C 180,E1 -21297.792,E2 -21297.792} C_VEL
LIN {X 0,Y 210.878,Z 416.168,A -85,B 0,C 180,E1 -21298.897,E2 -21298.897} C_VEL
LIN {X 0,Y 207.98,Z 426.606,A -85,B 0,C 180,E1 -21305.014,E2 -21305.014} C_VEL
LIN {X 0,Y 206.479,Z 435.848,A -85,B 0,C 180,E1 -21310.422,E2 -21310.422} C_VEL
LIN {X 0,Y 206.601,Z 448.03,A -85,B 0,C 180,E1 -21311.421,E2 -21311.421} C_VEL
LIN {X 0,Y 207.383,Z 460.852,A -85,B 0,C 180,E1 -21312.878,E2 -21312.878} C_VEL
LIN {X 0,Y 208.21,Z 470.885,A -85,B 0,C 180,E1 -21314.334,E2 -21314.334} C_VEL
LIN {X 0,Y 207.611,Z 481.201,A -85,B 0,C 180,E1 -21316.293,E2 -21316.293} C_VEL
LIN {X 0,Y 207.105,Z 491.516,A -85,B 0,C 180,E1 -21318.749,E2 -21318.749} C_VEL
LIN {X 0,Y 206.847,Z 499.428,A -85,B 0,C 180,E1 -21321.1,E2 -21321.1} C_VEL
LIN {X 0,Y 206.869,Z 506.757,A -85,B 0,C 180,E1 -21323.78,E2 -21323.78} C_VEL
LIN {X 0,Y 206.32,Z 509.78,A -85,B 0,C 180,E1 -21325.183,E2 -21325.183} C_VEL
LIN {X 0,Y 204.819,Z 512.22,A -85,B 0,C 180,E1 -21326.635,E2 -21326.635} C_VEL
LIN {X 0,Y 201.056,Z 516.053,A -85,B 0,C 180,E1 -21329.696,E2 -21329.696} C_VEL
LIN {X 0,Y 199.641,Z 518.353,A -85,B 0,C 180,E1 -21331.872,E2 -21331.872} C_VEL
LIN {X 0,Y 198.978,Z 520.335,A -85,B 0,C 180,E1 -21334.051,E2 -21334.051} C_VEL
LIN {X 0,Y 198.405,Z 522.368,A -85,B 0,C 180,E1 -21337.328,E2 -21337.328} C_VEL
LIN {X 0,Y 198.362,Z 523.332,A -85,B 0,C 180,E1 -21340.204,E2 -21340.204} C_VEL
LIN {X 0,Y 199.24,Z 523.59,A -85,B 0,C 180,E1 -21344.295,E2 -21344.295} C_VEL
LIN {X 0,Y 201.487,Z 522.5,A -85,B 0,C 180,E1 -21348.296,E2 -21348.296} C_VEL
LIN {X 0,Y 205.199,Z 519.911,A -85,B 0,C 180,E1 -21352.371,E2 -21352.371} C_VEL
LIN {X 0,Y 209.714,Z 516.294,A -85,B 0,C 180,E1 -21355.828,E2 -21355.828} C_VEL
LIN {X 0,Y 215.666,Z 511.01,A -85,B 0,C 180,E1 -21359.263,E2 -21359.263} C_VEL
LIN {X 0,Y 220.872,Z 505.973,A -85,B 0,C 180,E1 -21361.67,E2 -21361.67} C_VEL
LIN {X 0,Y 227.508,Z 498.789,A -85,B 0,C 180,E1 -21364.317,E2 -21364.317} C_VEL
LIN {X 0,Y 230.802,Z 494.281,A -85,B 0,C 180,E1 -21365.886,E2 -21365.886} C_VEL
LIN {X 0,Y 234.516,Z 487.952,A -85,B 0,C 180,E1 -21368.135,E2 -21368.135} C_VEL
LIN {X 0,Y 236.723,Z 483.719,A -85,B 0,C 180,E1 -21369.665,E2 -21369.665} C_VEL
LIN {X 0,Y 236.67,Z 482.053,A -85,B 0,C 180,E1 -21370.791,E2 -21370.791} C_VEL
LIN {X 0,Y 236.182,Z 478.32,A -85,B 0,C 180,E1 -21374.425,E2 -21374.425} C_VEL
LIN {X 0,Y 235.824,Z 476.87,A -85,B 0,C 180,E1 -21376.729,E2 -21376.729} C_VEL
LIN {X 0,Y 235.399,Z 476.293,A -85,B 0,C 180,E1 -21378.942,E2 -21378.942} C_VEL
LIN {X 0,Y 234.948,Z 476.435,A -85,B 0,C 180,E1 -21381.085,E2 -21381.085} C_VEL
LIN {X 0,Y 234.328,Z 477.522,A -85,B 0,C 180,E1 -21384.076,E2 -21384.076} C_VEL
LIN {X 0,Y 233.955,Z 478.285,A -85,B 0,C 180,E1 -21385.197,E2 -21385.197} C_VEL
LIN {X 0,Y 232.58,Z 480.777,A -85,B 0,C 180,E1 -21387.79,E2 -21387.79} C_VEL
LIN {X 0,Y 230.379,Z 484.341,A -85,B 0,C 180,E1 -21390.784,E2 -21390.784} C_VEL
LIN {X 0,Y 227.779,Z 487.722,A -85,B 0,C 180,E1 -21393.424,E2 -21393.424} C_VEL
LIN {X 0,Y 224.322,Z 490.374,A -85,B 0,C 180,E1 -21394.979,E2 -21394.979} C_VEL
LIN {X 0,Y 219.143,Z 493.584,A -85,B 0,C 180,E1 -21397.366,E2 -21397.366} C_VEL
LIN {X 0,Y 215.981,Z 495.072,A -85,B 0,C 180,E1 -21399.026,E2 -21399.026} C_VEL
LIN {X 0,Y 213.05,Z 496.046,A -85,B 0,C 180,E1 -21400.739,E2 -21400.739} C_VEL
LIN {X 0,Y 210.359,Z 496.564,A -85,B 0,C 180,E1 -21402.501,E2 -21402.501} C_VEL
LIN {X 0,Y 207.884,Z 496.561,A -85,B 0,C 180,E1 -21404.309,E2 -21404.309} C_VEL
LIN {X 0,Y 205.597,Z 496.067,A -85,B 0,C 180,E1 -21406.156,E2 -21406.156} C_VEL
LIN {X 0,Y 203.584,Z 495.059,A -85,B 0,C 180,E1 -21408.046,E2 -21408.046} C_VEL
LIN {X 0,Y 201.255,Z 492.523,A -85,B 0,C 180,E1 -21410.959,E2 -21410.959} C_VEL
LIN {X 0,Y 199.506,Z 488.793,A -85,B 0,C 180,E1 -21413.934,E2 -21413.934} C_VEL
LIN {X 0,Y 198.509,Z 483.682,A -85,B 0,C 180,E1 -21416.956,E2 -21416.956} C_VEL
LIN {X 0,Y 198.117,Z 477.118,A -85,B 0,C 180,E1 -21420,E2 -21420} C_VEL
LIN {X 0,Y 198.179,Z 470.238,A -85,B 0,C 180,E1 -21422.541,E2 -21422.541} C_VEL
LIN {X 0,Y 198.674,Z 461.834,A -85,B 0,C 180,E1 -21425.074,E2 -21425.074} C_VEL
LIN {X 0,Y 199.021,Z 451.262,A -85,B 0,C 180,E1 -21427.61,E2 -21427.61} C_VEL
LIN {X 0,Y 199.571,Z 440.178,A -85,B 0,C 180,E1 -21429.721,E2 -21429.721} C_VEL
LIN {X 0,Y 199.751,Z 434.244,A -85,B 0,C 180,E1 -21430.645,E2 -21430.645} C_VEL
LIN {X 0,Y 198.512,Z 422.391,A -85,B 0,C 180,E1 -21432.135,E2 -21432.135} C_VEL
LIN {X 0,Y 198.185,Z 417.894,A -85,B 0,C 180,E1 -21432.675,E2 -21432.675} C_VEL
LIN {X 0,Y 198.503,Z 410.929,A -85,B 0,C 180,E1 -21438.581,E2 -21438.581} C_VEL
LIN {X 0,Y 199.037,Z 405.398,A -85,B 0,C 180,E1 -21443.355,E2 -21443.355} C_VEL
LIN {X 0,Y 199.712,Z 399.673,A -85,B 0,C 180,E1 -21448.385,E2 -21448.385} C_VEL
LIN {X 0,Y 200.077,Z 395.882,A -85,B 0,C 180,E1 -21451.796,E2 -21451.796} C_VEL
LIN {X 0,Y 199.989,Z 395.563,A -85,B 0,C 180,E1 -21452.498,E2 -21452.498} C_VEL
LIN {X 0,Y 199.669,Z 395.613,A -85,B 0,C 180,E1 -21456.754,E2 -21456.754} C_VEL
LIN {X 0,Y 199.641,Z 395.616,A -85,B 0,C 180,E1 -21459.321,E2 -21459.321} C_VEL
LIN {X 0,Y 199.584,Z 395.623,A -85,B 0,C 180,E1 -21464.771,E2 -21464.771} C_VEL
LIN {X 0,Y 199.583,Z 395.623,A -85,B 0,C 180,E1 -21468.005,E2 -21468.005} C_VEL
LIN {X 0,Y 199.613,Z 395.617,A -85,B 0,C 180,E1 -21470.767,E2 -21470.767} C_VEL
LIN {X 0,Y 199.614,Z 395.619,A -85,B 0,C 180,E1 -21475.713,E2 -21475.713} C_VEL
LIN {X 0,Y 199.696,Z 395.609,A -85,B 0,C 180,E1 -21478.136,E2 -21478.136} C_VEL
LIN {X 0,Y 199.69,Z 395.611,A -85,B 0,C 180,E1 -21482.772,E2 -21482.772} C_VEL
LIN {X 0,Y 199.742,Z 395.6,A -85,B 0,C 180,E1 -21487.229,E2 -21487.229} C_VEL
LIN {X 0,Y 199.84,Z 395.59,A -85,B 0,C 180,E1 -21491.722,E2 -21491.722} C_VEL
LIN {X 0,Y 199.839,Z 395.59,A -85,B 0,C 180,E1 -21495.748,E2 -21495.748} C_VEL
LIN {X 0,Y 200.025,Z 395.568,A -85,B 0,C 180,E1 -21499.882,E2 -21499.882} C_VEL
LIN {X 0,Y 200.027,Z 395.569,A -85,B 0,C 180,E1 -21503.949,E2 -21503.949} C_VEL
LIN {X 0,Y 200.325,Z 395.531,A -85,B 0,C 180,E1 -21507.989,E2 -21507.989} C_VEL
LIN {X 0,Y 200.483,Z 395.514,A -85,B 0,C 180,E1 -21510,E2 -21510} C_VEL
LIN {X 0,Y 200.035,Z 395.565,A -85,B 0,C 180,E1 -21514.029,E2 -21514.029} C_VEL
LIN {X 0,Y 200.114,Z 395.559,A -85,B 0,C 180,E1 -21518.075,E2 -21518.075} C_VEL
LIN {X 0,Y 199.917,Z 395.578,A -85,B 0,C 180,E1 -21522.177,E2 -21522.177} C_VEL
LIN {X 0,Y 199.809,Z 395.595,A -85,B 0,C 180,E1 -21526.343,E2 -21526.343} C_VEL
LIN {X 0,Y 199.745,Z 395.599,A -85,B 0,C 180,E1 -21530.6,E2 -21530.6} C_VEL
LIN {X 0,Y 199.678,Z 395.611,A -85,B 0,C 180,E1 -21534.984,E2 -21534.984} C_VEL
LIN {X 0,Y 199.677,Z 395.609,A -85,B 0,C 180,E1 -21539.522,E2 -21539.522} C_VEL
LIN {X 0,Y 199.666,Z 395.611,A -85,B 0,C 180,E1 -21542.352,E2 -21542.352} C_VEL
LIN {X 0,Y 199.642,Z 395.615,A -85,B 0,C 180,E1 -21546.759,E2 -21546.759} C_VEL
LIN {X 0,Y 199.64,Z 395.614,A -85,B 0,C 180,E1 -21549.321,E2 -21549.321} C_VEL
LIN {X 0,Y 199.579,Z 395.624,A -85,B 0,C 180,E1 -21554.772,E2 -21554.772} C_VEL
LIN {X 0,Y 199.579,Z 395.62,A -85,B 0,C 180,E1 -21558.004,E2 -21558.004} C_VEL
LIN {X 0,Y 199.612,Z 395.62,A -85,B 0,C 180,E1 -21560.767,E2 -21560.767} C_VEL
LIN {X 0,Y 199.614,Z 395.615,A -85,B 0,C 180,E1 -21565.713,E2 -21565.713} C_VEL
LIN {X 0,Y 199.702,Z 395.607,A -85,B 0,C 180,E1 -21568.137,E2 -21568.137} C_VEL
LIN {X 0,Y 199.689,Z 395.61,A -85,B 0,C 180,E1 -21572.772,E2 -21572.772} C_VEL
LIN {X 0,Y 199.74,Z 395.604,A -85,B 0,C 180,E1 -21577.229,E2 -21577.229} C_VEL
LIN {X 0,Y 199.839,Z 395.588,A -85,B 0,C 180,E1 -21581.722,E2 -21581.722} C_VEL
LIN {X 0,Y 199.85,Z 395.589,A -85,B 0,C 180,E1 -21585.749,E2 -21585.749} C_VEL
LIN {X 0,Y 200.077,Z 395.559,A -85,B 0,C 180,E1 -21589.884,E2 -21589.884} C_VEL
LIN {X 0,Y 200.134,Z 395.55,A -85,B 0,C 180,E1 -21591.925,E2 -21591.925} C_VEL
LIN {X 0,Y 200.324,Z 395.53,A -85,B 0,C 180,E1 -21597.989,E2 -21597.989} C_VEL
LIN {X 0,Y 200.482,Z 395.508,A -85,B 0,C 180,E1 -21600,E2 -21600} C_VEL
LIN {X 0,Y 200.038,Z 395.567,A -85,B 0,C 180,E1 -21604.029,E2 -21604.029} C_VEL
LIN {X 0,Y 200.134,Z 395.553,A -85,B 0,C 180,E1 -21608.075,E2 -21608.075} C_VEL
LIN {X 0,Y 199.916,Z 395.583,A -85,B 0,C 180,E1 -21612.177,E2 -21612.177} C_VEL
LIN {X 0,Y 199.807,Z 395.593,A -85,B 0,C 180,E1 -21616.343,E2 -21616.343} C_VEL
LIN {X 0,Y 199.702,Z 395.609,A -85,B 0,C 180,E1 -21620.605,E2 -21620.605} C_VEL
LIN {X 0,Y 199.674,Z 395.608,A -85,B 0,C 180,E1 -21624.984,E2 -21624.984} C_VEL
LIN {X 0,Y 199.666,Z 395.613,A -85,B 0,C 180,E1 -21629.524,E2 -21629.524} C_VEL
LIN {X 0,Y 199.659,Z 395.612,A -85,B 0,C 180,E1 -21632.349,E2 -21632.349} C_VEL
LIN {X 0,Y 199.641,Z 395.615,A -85,B 0,C 180,E1 -21636.759,E2 -21636.759} C_VEL
LIN {X 0,Y 199.64,Z 395.616,A -85,B 0,C 180,E1 -21639.321,E2 -21639.321} C_VEL
LIN {X 0,Y 199.767,Z 395.743,A -85,B 0,C 180,E1 -21645.282,E2 -21645.282} C_VEL
LIN {X 0,Y 201.151,Z 403.009,A -85,B 0,C 180,E1 -21650.233,E2 -21650.233} C_VEL
LIN {X 0,Y 202.805,Z 410.435,A -85,B 0,C 180,E1 -21655.056,E2 -21655.056} C_VEL
LIN {X 0,Y 203.821,Z 414.582,A -85,B 0,C 180,E1 -21657.693,E2 -21657.693} C_VEL
LIN {X 0,Y 203.723,Z 416.428,A -85,B 0,C 180,E1 -21658.837,E2 -21658.837} C_VEL
LIN {X 0,Y 200.8,Z 426.755,A -85,B 0,C 180,E1 -21665.166,E2 -21665.166} C_VEL
LIN {X 0,Y 199.433,Z 435.27,A -85,B 0,C 180,E1 -21670.508,E2 -21670.508} C_VEL
LIN {X 0,Y 199.574,Z 448.708,A -85,B 0,C 180,E1 -21671.701,E2 -21671.701} C_VEL
LIN {X 0,Y 200.385,Z 461.02,A -85,B 0,C 180,E1 -21673.181,E2 -21673.181} C_VEL
LIN {X 0,Y 201.159,Z 471.523,A -85,B 0,C 180,E1 -21674.809,E2 -21674.809} C_VEL
LIN {X 0,Y 200.538,Z 481.526,A -85,B 0,C 180,E1 -21676.833,E2 -21676.833} C_VEL
LIN {X 0,Y 200.16,Z 490.995,A -85,B 0,C 180,E1 -21679.211,E2 -21679.211} C_VEL
LIN {X 0,Y 199.922,Z 499.614,A -85,B 0,C 180,E1 -21681.917,E2 -21681.917} C_VEL
LIN {X 0,Y 200.093,Z 507.327,A -85,B 0,C 180,E1 -21684.963,E2 -21684.963} C_VEL
LIN {X 0,Y 200.123,Z 513.143,A -85,B 0,C 180,E1 -21687.988,E2 -21687.988} C_VEL
LIN {X 0,Y 199.84,Z 517.42,A -85,B 0,C 180,E1 -21691.008,E2 -21691.008} C_VEL
LIN {X 0,Y 199.641,Z 518.353,A -85,B 0,C 180,E1 -21691.872,E2 -21691.872} C_VEL
LIN {X 0,Y 198.624,Z 519.799,A -85,B 0,C 180,E1 -21693.489,E2 -21693.489} C_VEL
LIN {X 0,Y 196.698,Z 520.731,A -85,B 0,C 180,E1 -21695.098,E2 -21695.098} C_VEL
LIN {X 0,Y 192.529,Z 521.648,A -85,B 0,C 180,E1 -21698.408,E2 -21698.408} C_VEL
LIN {X 0,Y 191.477,Z 521.945,A -85,B 0,C 180,E1 -21700.163,E2 -21700.163} C_VEL
LIN {X 0,Y 191.438,Z 522.058,A -85,B 0,C 180,E1 -21700.759,E2 -21700.759} C_VEL
LIN {X 0,Y 192.39,Z 522.562,A -85,B 0,C 180,E1 -21704.816,E2 -21704.816} C_VEL
LIN {X 0,Y 194.738,Z 521.859,A -85,B 0,C 180,E1 -21708.954,E2 -21708.954} C_VEL
LIN {X 0,Y 198.409,Z 519.823,A -85,B 0,C 180,E1 -21712.932,E2 -21712.932} C_VEL
LIN {X 0,Y 203.349,Z 516.465,A -85,B 0,C 180,E1 -21716.699,E2 -21716.699} C_VEL
LIN {X 0,Y 209.531,Z 511.682,A -85,B 0,C 180,E1 -21720.207,E2 -21720.207} C_VEL
LIN {X 0,Y 216.868,Z 505.318,A -85,B 0,C 180,E1 -21723.43,E2 -21723.43} C_VEL
LIN {X 0,Y 222.788,Z 499.426,A -85,B 0,C 180,E1 -21725.704,E2 -21725.704} C_VEL
LIN {X 0,Y 226.882,Z 494.166,A -85,B 0,C 180,E1 -21727.719,E2 -21727.719} C_VEL
LIN {X 0,Y 230.452,Z 488.703,A -85,B 0,C 180,E1 -21729.824,E2 -21729.824} C_VEL
LIN {X 0,Y 231.186,Z 487.179,A -85,B 0,C 180,E1 -21730.536,E2 -21730.536} C_VEL
LIN {X 0,Y 231.012,Z 484.368,A -85,B 0,C 180,E1 -21733.102,E2 -21733.102} C_VEL
LIN {X 0,Y 230.841,Z 482.403,A -85,B 0,C 180,E1 -21735.554,E2 -21735.554} C_VEL
LIN {X 0,Y 230.469,Z 481.396,A -85,B 0,C 180,E1 -21737.865,E2 -21737.865} C_VEL
LIN {X 0,Y 229.919,Z 481.202,A -85,B 0,C 180,E1 -21740.065,E2 -21740.065} C_VEL
LIN {X 0,Y 229.242,Z 481.68,A -85,B 0,C 180,E1 -21742.854,E2 -21742.854} C_VEL
LIN {X 0,Y 228.777,Z 482.327,A -85,B 0,C 180,E1 -21744.29,E2 -21744.29} C_VEL
LIN {X 0,Y 227.62,Z 483.927,A -85,B 0,C 180,E1 -21746.476,E2 -21746.476} C_VEL
LIN {X 0,Y 226.333,Z 485.499,A -85,B 0,C 180,E1 -21748.138,E2 -21748.138} C_VEL
LIN {X 0,Y 224.748,Z 487.439,A -85,B 0,C 180,E1 -21749.978,E2 -21749.978} C_VEL
LIN {X 0,Y 222.384,Z 489.88,A -85,B 0,C 180,E1 -21752.238,E2 -21752.238} C_VEL
LIN {X 0,Y 219.782,Z 491.779,A -85,B 0,C 180,E1 -21753.555,E2 -21753.555} C_VEL
LIN {X 0,Y 216.299,Z 493.777,A -85,B 0,C 180,E1 -21755.014,E2 -21755.014} C_VEL
LIN {X 0,Y 212.806,Z 495.466,A -85,B 0,C 180,E1 -21756.653,E2 -21756.653} C_VEL
LIN {X 0,Y 209.516,Z 496.674,A -85,B 0,C 180,E1 -21758.347,E2 -21758.347} C_VEL
LIN {X 0,Y 206.466,Z 497.38,A -85,B 0,C 180,E1 -21760.099,E2 -21760.099} C_VEL
LIN {X 0,Y 203.668,Z 497.621,A -85,B 0,C 180,E1 -21761.907,E2 -21761.907} C_VEL
LIN {X 0,Y 201.11,Z 497.356,A -85,B 0,C 180,E1 -21763.766,E2 -21763.766} C_VEL
LIN {X 0,Y 198.722,Z 496.617,A -85,B 0,C 180,E1 -21765.667,E2 -21765.667} C_VEL
LIN {X 0,Y 196.657,Z 495.34,A -85,B 0,C 180,E1 -21767.618,E2 -21767.618} C_VEL
LIN {X 0,Y 194.256,Z 492.45,A -85,B 0,C 180,E1 -21770.63,E2 -21770.63} C_VEL
LIN {X 0,Y 192.455,Z 488.332,A -85,B 0,C 180,E1 -21773.711,E2 -21773.711} C_VEL
LIN {X 0,Y 191.477,Z 482.872,A -85,B 0,C 180,E1 -21776.844,E2 -21776.844} C_VEL
LIN {X 0,Y 191.09,Z 475.854,A -85,B 0,C 180,E1 -21780,E2 -21780} C_VEL
LIN {X 0,Y 191.195,Z 468.654,A -85,B 0,C 180,E1 -21782.634,E2 -21782.634} C_VEL
LIN {X 0,Y 191.685,Z 459.766,A -85,B 0,C 180,E1 -21785.259,E2 -21785.259} C_VEL
LIN {X 0,Y 192.028,Z 449.738,A -85,B 0,C 180,E1 -21787.624,E2 -21787.624} C_VEL
LIN {X 0,Y 192.527,Z 439.082,A -85,B 0,C 180,E1 -21789.647,E2 -21789.647} C_VEL
LIN {X 0,Y 192.617,Z 433.636,A -85,B 0,C 180,E1 -21790.512,E2 -21790.512} C_VEL
LIN {X 0,Y 191.368,Z 421.533,A -85,B 0,C 180,E1 -21792.057,E2 -21792.057} C_VEL
LIN {X 0,Y 191.129,Z 418.244,A -85,B 0,C 180,E1 -21792.476,E2 -21792.476} C_VEL
LIN {X 0,Y 191.338,Z 411.826,A -85,B 0,C 180,E1 -21798.082,E2 -21798.082} C_VEL
LIN {X 0,Y 191.86,Z 406.71,A -85,B 0,C 180,E1 -21802.621,E2 -21802.621} C_VEL
LIN {X 0,Y 192.602,Z 400.401,A -85,B 0,C 180,E1 -21808.318,E2 -21808.318} C_VEL
LIN {X 0,Y 193.03,Z 396.515,A -85,B 0,C 180,E1 -21811.91,E2 -21811.91} C_VEL
LIN {X 0,Y 192.584,Z 396.495,A -85,B 0,C 180,E1 -21818.345,E2 -21818.345} C_VEL
LIN {X 0,Y 192.495,Z 396.504,A -85,B 0,C 180,E1 -21823.096,E2 -21823.096} C_VEL
LIN {X 0,Y 192.515,Z 396.505,A -85,B 0,C 180,E1 -21826.897,E2 -21826.897} C_VEL
LIN {X 0,Y 192.554,Z 396.494,A -85,B 0,C 180,E1 -21831.648,E2 -21831.648} C_VEL
LIN {X 0,Y 192.599,Z 396.494,A -85,B 0,C 180,E1 -21836.814,E2 -21836.814} C_VEL
LIN {X 0,Y 192.667,Z 396.482,A -85,B 0,C 180,E1 -21841.692,E2 -21841.692} C_VEL
LIN {X 0,Y 192.709,Z 396.48,A -85,B 0,C 180,E1 -21846.349,E2 -21846.349} C_VEL
LIN {X 0,Y 192.784,Z 396.469,A -85,B 0,C 180,E1 -21851.414,E2 -21851.414} C_VEL
LIN {X 0,Y 192.768,Z 396.47,A -85,B 0,C 180,E1 -21855.214,E2 -21855.214} C_VEL
LIN {X 0,Y 192.948,Z 396.448,A -85,B 0,C 180,E1 -21859.566,E2 -21859.566} C_VEL
LIN {X 0,Y 192.989,Z 396.445,A -85,B 0,C 180,E1 -21863.728,E2 -21863.728} C_VEL
LIN {X 0,Y 193.266,Z 396.41,A -85,B 0,C 180,E1 -21867.916,E2 -21867.916} C_VEL
LIN {X 0,Y 193.447,Z 396.39,A -85,B 0,C 180,E1 -21870,E2 -21870} C_VEL
LIN {X 0,Y 192.981,Z 396.443,A -85,B 0,C 180,E1 -21874.177,E2 -21874.177} C_VEL
LIN {X 0,Y 193.065,Z 396.435,A -85,B 0,C 180,E1 -21878.372,E2 -21878.372} C_VEL
LIN {X 0,Y 192.856,Z 396.456,A -85,B 0,C 180,E1 -21882.63,E2 -21882.63} C_VEL
LIN {X 0,Y 192.784,Z 396.469,A -85,B 0,C 180,E1 -21888.587,E2 -21888.587} C_VEL
LIN {X 0,Y 192.671,Z 396.484,A -85,B 0,C 180,E1 -21894.227,E2 -21894.227} C_VEL
LIN {X 0,Y 192.652,Z 396.484,A -85,B 0,C 180,E1 -21898.892,E2 -21898.892} C_VEL
LIN {X 0,Y 192.602,Z 396.493,A -85,B 0,C 180,E1 -21903.185,E2 -21903.185} C_VEL
LIN {X 0,Y 192.611,Z 396.49,A -85,B 0,C 180,E1 -21906.607,E2 -21906.607} C_VEL
LIN {X 0,Y 192.524,Z 396.502,A -85,B 0,C 180,E1 -21911.078,E2 -21911.078} C_VEL
LIN {X 0,Y 192.491,Z 396.503,A -85,B 0,C 180,E1 -21916.075,E2 -21916.075} C_VEL
LIN {X 0,Y 192.519,Z 396.502,A -85,B 0,C 180,E1 -21920.051,E2 -21920.051} C_VEL
LIN {X 0,Y 192.562,Z 396.495,A -85,B 0,C 180,E1 -21924.27,E2 -21924.27} C_VEL
LIN {X 0,Y 192.612,Z 396.49,A -85,B 0,C 180,E1 -21927.058,E2 -21927.058} C_VEL
LIN {X 0,Y 192.666,Z 396.483,A -85,B 0,C 180,E1 -21931.692,E2 -21931.692} C_VEL
LIN {X 0,Y 192.708,Z 396.478,A -85,B 0,C 180,E1 -21936.349,E2 -21936.349} C_VEL
LIN {X 0,Y 192.783,Z 396.467,A -85,B 0,C 180,E1 -21941.414,E2 -21941.414} C_VEL
LIN {X 0,Y 192.856,Z 396.461,A -85,B 0,C 180,E1 -21947.37,E2 -21947.37} C_VEL
LIN {X 0,Y 193.081,Z 396.428,A -85,B 0,C 180,E1 -21951.628,E2 -21951.628} C_VEL
LIN {X 0,Y 193.266,Z 396.409,A -85,B 0,C 180,E1 -21957.916,E2 -21957.916} C_VEL
LIN {X 0,Y 193.446,Z 396.384,A -85,B 0,C 180,E1 -21960,E2 -21960} C_VEL
LIN {X 0,Y 192.985,Z 396.446,A -85,B 0,C 180,E1 -21964.177,E2 -21964.177} C_VEL
LIN {X 0,Y 193.081,Z 396.431,A -85,B 0,C 180,E1 -21968.372,E2 -21968.372} C_VEL
LIN {X 0,Y 192.855,Z 396.462,A -85,B 0,C 180,E1 -21972.63,E2 -21972.63} C_VEL
LIN {X 0,Y 192.759,Z 396.468,A -85,B 0,C 180,E1 -21976.958,E2 -21976.958} C_VEL
LIN {X 0,Y 192.638,Z 396.488,A -85,B 0,C 180,E1 -21981.397,E2 -21981.397} C_VEL
LIN {X 0,Y 192.665,Z 396.483,A -85,B 0,C 180,E1 -21984.225,E2 -21984.225} C_VEL
LIN {X 0,Y 192.645,Z 396.487,A -85,B 0,C 180,E1 -21988.889,E2 -21988.889} C_VEL
LIN {X 0,Y 192.599,Z 396.49,A -85,B 0,C 180,E1 -21993.186,E2 -21993.186} C_VEL
LIN {X 0,Y 192.61,Z 396.491,A -85,B 0,C 180,E1 -21996.607,E2 -21996.607} C_VEL
LIN {X 0,Y 192.529,Z 396.5,A -85,B 0,C 180,E1 -22001.076,E2 -22001.076} C_VEL
LIN {X 0,Y 192.681,Z 396.576,A -85,B 0,C 180,E1 -22005.089,E2 -22005.089} C_VEL
LIN {X 0,Y 193.902,Z 402.875,A -85,B 0,C 180,E1 -22009.566,E2 -22009.566} C_VEL
LIN {X 0,Y 195.266,Z 408.984,A -85,B 0,C 180,E1 -22013.729,E2 -22013.729} C_VEL
LIN {X 0,Y 196.667,Z 414.807,A -85,B 0,C 180,E1 -22017.586,E2 -22017.586} C_VEL
LIN {X 0,Y 196.333,Z 417.347,A -85,B 0,C 180,E1 -22019.217,E2 -22019.217} C_VEL
LIN {X 0,Y 193.465,Z 427.503,A -85,B 0,C 180,E1 -22025.755,E2 -22025.755} C_VEL
LIN {X 0,Y 192.371,Z 434.969,A -85,B 0,C 180,E1 -22030.665,E2 -22030.665} C_VEL
LIN {X 0,Y 192.522,Z 448.14,A -85,B 0,C 180,E1 -22031.896,E2 -22031.896} C_VEL
LIN {X 0,Y 193.388,Z 460.943,A -85,B 0,C 180,E1 -22033.506,E2 -22033.506} C_VEL
LIN {X 0,Y 194.18,Z 470.573,A -85,B 0,C 180,E1 -22035.056,E2 -22035.056} C_VEL
LIN {X 0,Y 193.6,Z 480.588,A -85,B 0,C 180,E1 -22037.153,E2 -22037.153} C_VEL
LIN {X 0,Y 193.263,Z 489.744,A -85,B 0,C 180,E1 -22039.524,E2 -22039.524} C_VEL
LIN {X 0,Y 193.078,Z 497.888,A -85,B 0,C 180,E1 -22042.155,E2 -22042.155} C_VEL
LIN {X 0,Y 193.274,Z 505.754,A -85,B 0,C 180,E1 -22045.307,E2 -22045.307} C_VEL
LIN {X 0,Y 193.304,Z 510.816,A -85,B 0,C 180,E1 -22047.917,E2 -22047.917} C_VEL
LIN {X 0,Y 193.206,Z 514.044,A -85,B 0,C 180,E1 -22050,E2 -22050} C_VEL
LIN {X 0,Y 192.772,Z 516.622,A -85,B 0,C 180,E1 -22052.09,E2 -22052.09} C_VEL
LIN {X 0,Y 191.671,Z 520.063,A -85,B 0,C 180,E1 -22056.316,E2 -22056.316} C_VEL
LIN {X 0,Y 191.438,Z 522.058,A -85,B 0,C 180,E1 -22060.759,E2 -22060.759} C_VEL
LIN {X 0,Y 191.052,Z 522.312,A -85,B 0,C 180,E1 -22062.525,E2 -22062.525} C_VEL
LIN {X 0,Y 189.126,Z 522.089,A -85,B 0,C 180,E1 -22065.46,E2 -22065.46} C_VEL
LIN {X 0,Y 187.855,Z 521.441,A -85,B 0,C 180,E1 -22068.436,E2 -22068.436} C_VEL
LIN {X 0,Y 188.486,Z 520.916,A -85,B 0,C 180,E1 -22070.212,E2 -22070.212} C_VEL
LIN {X 0,Y 191.883,Z 519.445,A -85,B 0,C 180,E1 -22073.759,E2 -22073.759} C_VEL
LIN {X 0,Y 197.047,Z 516.552,A -85,B 0,C 180,E1 -22077.624,E2 -22077.624} C_VEL
LIN {X 0,Y 203.462,Z 512.237,A -85,B 0,C 180,E1 -22081.207,E2 -22081.207} C_VEL
LIN {X 0,Y 209.046,Z 508.058,A -85,B 0,C 180,E1 -22083.692,E2 -22083.692} C_VEL
LIN {X 0,Y 215.175,Z 502.917,A -85,B 0,C 180,E1 -22086.009,E2 -22086.009} C_VEL
LIN {X 0,Y 219.057,Z 499.157,A -85,B 0,C 180,E1 -22087.559,E2 -22087.559} C_VEL
LIN {X 0,Y 223.823,Z 493.248,A -85,B 0,C 180,E1 -22090.045,E2 -22090.045} C_VEL
LIN {X 0,Y 225.286,Z 491.25,A -85,B 0,C 180,E1 -22090.929,E2 -22090.929} C_VEL
LIN {X 0,Y 225.49,Z 490.404,A -85,B 0,C 180,E1 -22091.58,E2 -22091.58} C_VEL
LIN {X 0,Y 225.47,Z 487.969,A -85,B 0,C 180,E1 -22094.199,E2 -22094.199} C_VEL
LIN {X 0,Y 225.239,Z 486.434,A -85,B 0,C 180,E1 -22096.65,E2 -22096.65} C_VEL
LIN {X 0,Y 224.692,Z 485.816,A -85,B 0,C 180,E1 -22098.94,E2 -22098.94} C_VEL
LIN {X 0,Y 223.931,Z 485.87,A -85,B 0,C 180,E1 -22101.686,E2 -22101.686} C_VEL
LIN {X 0,Y 223.441,Z 486.26,A -85,B 0,C 180,E1 -22103.301,E2 -22103.301} C_VEL
LIN {X 0,Y 222.296,Z 487.31,A -85,B 0,C 180,E1 -22105.314,E2 -22105.314} C_VEL
LIN {X 0,Y 220.844,Z 488.764,A -85,B 0,C 180,E1 -22107.248,E2 -22107.248} C_VEL
LIN {X 0,Y 219.074,Z 490.364,A -85,B 0,C 180,E1 -22109.117,E2 -22109.117} C_VEL
LIN {X 0,Y 217.091,Z 492.022,A -85,B 0,C 180,E1 -22110.948,E2 -22110.948} C_VEL
LIN {X 0,Y 213.977,Z 493.963,A -85,B 0,C 180,E1 -22112.624,E2 -22112.624} C_VEL
LIN {X 0,Y 210.102,Z 495.847,A -85,B 0,C 180,E1 -22114.224,E2 -22114.224} C_VEL
LIN {X 0,Y 206.467,Z 497.244,A -85,B 0,C 180,E1 -22115.891,E2 -22115.891} C_VEL
LIN {X 0,Y 203.065,Z 498.13,A -85,B 0,C 180,E1 -22117.623,E2 -22117.623} C_VEL
LIN {X 0,Y 199.881,Z 498.59,A -85,B 0,C 180,E1 -22119.414,E2 -22119.414} C_VEL
LIN {X 0,Y 196.975,Z 498.547,A -85,B 0,C 180,E1 -22121.27,E2 -22121.27} C_VEL
LIN {X 0,Y 194.318,Z 498.025,A -85,B 0,C 180,E1 -22123.182,E2 -22123.182} C_VEL
LIN {X 0,Y 191.866,Z 497.015,A -85,B 0,C 180,E1 -22125.143,E2 -22125.143} C_VEL
LIN {X 0,Y 188.838,Z 494.522,A -85,B 0,C 180,E1 -22128.189,E2 -22128.189} C_VEL
LIN {X 0,Y 186.533,Z 490.871,A -85,B 0,C 180,E1 -22131.332,E2 -22131.332} C_VEL
LIN {X 0,Y 184.997,Z 485.917,A -85,B 0,C 180,E1 -22134.55,E2 -22134.55} C_VEL
LIN {X 0,Y 184.252,Z 479.619,A -85,B 0,C 180,E1 -22137.814,E2 -22137.814} C_VEL
LIN {X 0,Y 184.089,Z 471.546,A -85,B 0,C 180,E1 -22141.094,E2 -22141.094} C_VEL
LIN {X 0,Y 184.426,Z 463.268,A -85,B 0,C 180,E1 -22143.824,E2 -22143.824} C_VEL
LIN {X 0,Y 184.784,Z 454.144,A -85,B 0,C 180,E1 -22146.278,E2 -22146.278} C_VEL
LIN {X 0,Y 185.233,Z 444.053,A -85,B 0,C 180,E1 -22148.455,E2 -22148.455} C_VEL
LIN {X 0,Y 185.638,Z 434.275,A -85,B 0,C 180,E1 -22150.156,E2 -22150.156} C_VEL
LIN {X 0,Y 184.313,Z 421.613,A -85,B 0,C 180,E1 -22151.827,E2 -22151.827} C_VEL
LIN {X 0,Y 184.091,Z 418.643,A -85,B 0,C 180,E1 -22152.191,E2 -22152.191} C_VEL
LIN {X 0,Y 184.321,Z 411.21,A -85,B 0,C 180,E1 -22158.911,E2 -22158.911} C_VEL
LIN {X 0,Y 184.961,Z 405.434,A -85,B 0,C 180,E1 -22164.225,E2 -22164.225} C_VEL
LIN {X 0,Y 185.718,Z 399.798,A -85,B 0,C 180,E1 -22169.497,E2 -22169.497} C_VEL
LIN {X 0,Y 185.972,Z 397.313,A -85,B 0,C 180,E1 -22171.943,E2 -22171.943} C_VEL
LIN {X 0,Y 185.57,Z 397.369,A -85,B 0,C 180,E1 -22177.314,E2 -22177.314} C_VEL
LIN {X 0,Y 185.486,Z 397.38,A -85,B 0,C 180,E1 -22180.73,E2 -22180.73} C_VEL
LIN {X 0,Y 185.465,Z 397.381,A -85,B 0,C 180,E1 -22186.054,E2 -22186.054} C_VEL
LIN {X 0,Y 185.471,Z 397.379,A -85,B 0,C 180,E1 -22189.896,E2 -22189.896} C_VEL
LIN {X 0,Y 185.509,Z 397.375,A -85,B 0,C 180,E1 -22192.711,E2 -22192.711} C_VEL
LIN {X 0,Y 185.545,Z 397.371,A -85,B 0,C 180,E1 -22197.975,E2 -22197.975} C_VEL
LIN {X 0,Y 185.584,Z 397.365,A -85,B 0,C 180,E1 -22200.576,E2 -22200.576} C_VEL
LIN {X 0,Y 185.59,Z 397.365,A -85,B 0,C 180,E1 -22205.383,E2 -22205.383} C_VEL
LIN {X 0,Y 185.697,Z 397.352,A -85,B 0,C 180,E1 -22211.115,E2 -22211.115} C_VEL
LIN {X 0,Y 185.702,Z 397.351,A -85,B 0,C 180,E1 -22214.638,E2 -22214.638} C_VEL
LIN {X 0,Y 185.891,Z 397.327,A -85,B 0,C 180,E1 -22219.418,E2 -22219.418} C_VEL
LIN {X 0,Y 185.951,Z 397.32,A -85,B 0,C 180,E1 -22223.489,E2 -22223.489} C_VEL
LIN {X 0,Y 186.21,Z 397.288,A -85,B 0,C 180,E1 -22227.837,E2 -22227.837} C_VEL
LIN {X 0,Y 186.41,Z 397.267,A -85,B 0,C 180,E1 -22230,E2 -22230} C_VEL
LIN {X 0,Y 185.929,Z 397.321,A -85,B 0,C 180,E1 -22234.335,E2 -22234.335} C_VEL
LIN {X 0,Y 186.012,Z 397.313,A -85,B 0,C 180,E1 -22238.692,E2 -22238.692} C_VEL
LIN {X 0,Y 185.768,Z 397.339,A -85,B 0,C 180,E1 -22243.12,E2 -22243.12} C_VEL
LIN {X 0,Y 185.72,Z 397.352,A -85,B 0,C 180,E1 -22247.622,E2 -22247.622} C_VEL
LIN {X 0,Y 185.619,Z 397.36,A -85,B 0,C 180,E1 -22252.248,E2 -22252.248} C_VEL
LIN {X 0,Y 185.566,Z 397.369,A -85,B 0,C 180,E1 -22257.031,E2 -22257.031} C_VEL
LIN {X 0,Y 185.581,Z 397.365,A -85,B 0,C 180,E1 -22259.493,E2 -22259.493} C_VEL
LIN {X 0,Y 185.521,Z 397.374,A -85,B 0,C 180,E1 -22264.627,E2 -22264.627} C_VEL
LIN {X 0,Y 185.545,Z 397.37,A -85,B 0,C 180,E1 -22267.304,E2 -22267.304} C_VEL
LIN {X 0,Y 185.486,Z 397.377,A -85,B 0,C 180,E1 -22270.729,E2 -22270.729} C_VEL
LIN {X 0,Y 185.46,Z 397.379,A -85,B 0,C 180,E1 -22276.055,E2 -22276.055} C_VEL
LIN {X 0,Y 185.469,Z 397.381,A -85,B 0,C 180,E1 -22279.895,E2 -22279.895} C_VEL
LIN {X 0,Y 185.508,Z 397.377,A -85,B 0,C 180,E1 -22282.711,E2 -22282.711} C_VEL
LIN {X 0,Y 185.548,Z 397.37,A -85,B 0,C 180,E1 -22287.975,E2 -22287.975} C_VEL
LIN {X 0,Y 185.583,Z 397.368,A -85,B 0,C 180,E1 -22290.576,E2 -22290.576} C_VEL
LIN {X 0,Y 185.589,Z 397.365,A -85,B 0,C 180,E1 -22295.382,E2 -22295.382} C_VEL
LIN {X 0,Y 185.696,Z 397.351,A -85,B 0,C 180,E1 -22301.115,E2 -22301.115} C_VEL
LIN {X 0,Y 185.73,Z 397.348,A -85,B 0,C 180,E1 -22304.64,E2 -22304.64} C_VEL
LIN {X 0,Y 185.944,Z 397.32,A -85,B 0,C 180,E1 -22309.328,E2 -22309.328} C_VEL
LIN {X 0,Y 185.971,Z 397.317,A -85,B 0,C 180,E1 -22313.49,E2 -22313.49} C_VEL
LIN {X 0,Y 186.21,Z 397.288,A -85,B 0,C 180,E1 -22317.837,E2 -22317.837} C_VEL
LIN {X 0,Y 186.409,Z 397.26,A -85,B 0,C 180,E1 -22320,E2 -22320} C_VEL
LIN {X 0,Y 185.932,Z 397.326,A -85,B 0,C 180,E1 -22324.335,E2 -22324.335} C_VEL
LIN {X 0,Y 186.031,Z 397.309,A -85,B 0,C 180,E1 -22328.691,E2 -22328.691} C_VEL
LIN {X 0,Y 185.767,Z 397.344,A -85,B 0,C 180,E1 -22333.12,E2 -22333.12} C_VEL
LIN {X 0,Y 185.692,Z 397.349,A -85,B 0,C 180,E1 -22337.625,E2 -22337.625} C_VEL
LIN {X 0,Y 185.598,Z 397.366,A -85,B 0,C 180,E1 -22342.251,E2 -22342.251} C_VEL
LIN {X 0,Y 185.562,Z 397.367,A -85,B 0,C 180,E1 -22347.032,E2 -22347.032} C_VEL
LIN {X 0,Y 185.578,Z 397.368,A -85,B 0,C 180,E1 -22349.493,E2 -22349.493} C_VEL
LIN {X 0,Y 185.519,Z 397.371,A -85,B 0,C 180,E1 -22354.628,E2 -22354.628} C_VEL
LIN {X 0,Y 185.544,Z 397.371,A -85,B 0,C 180,E1 -22357.304,E2 -22357.304} C_VEL
LIN {X 0,Y 185.505,Z 397.371,A -85,B 0,C 180,E1 -22362.996,E2 -22362.996} C_VEL
LIN {X 0,Y 185.652,Z 397.515,A -85,B 0,C 180,E1 -22365.003,E2 -22365.003} C_VEL
LIN {X 0,Y 187.082,Z 404.727,A -85,B 0,C 180,E1 -22370.31,E2 -22370.31} C_VEL
LIN {X 0,Y 188.61,Z 411.47,A -85,B 0,C 180,E1 -22375.061,E2 -22375.061} C_VEL
LIN {X 0,Y 189.504,Z 414.965,A -85,B 0,C 180,E1 -22377.471,E2 -22377.471} C_VEL
LIN {X 0,Y 189.403,Z 416.808,A -85,B 0,C 180,E1 -22378.702,E2 -22378.702} C_VEL
LIN {X 0,Y 186.804,Z 425.505,A -85,B 0,C 180,E1 -22384.547,E2 -22384.547} C_VEL
LIN {X 0,Y 185.337,Z 434.683,A -85,B 0,C 180,E1 -22390.878,E2 -22390.878} C_VEL
LIN {X 0,Y 185.505,Z 448.129,A -85,B 0,C 180,E1 -22392.211,E2 -22392.211} C_VEL
LIN {X 0,Y 186.382,Z 460.567,A -85,B 0,C 180,E1 -22393.854,E2 -22393.854} C_VEL
LIN {X 0,Y 187.206,Z 469.403,A -85,B 0,C 180,E1 -22395.321,E2 -22395.321} C_VEL
LIN {X 0,Y 186.698,Z 479.669,A -85,B 0,C 180,E1 -22397.555,E2 -22397.555} C_VEL
LIN {X 0,Y 186.386,Z 488.871,A -85,B 0,C 180,E1 -22400.029,E2 -22400.029} C_VEL
LIN {X 0,Y 186.234,Z 497.546,A -85,B 0,C 180,E1 -22402.955,E2 -22402.955} C_VEL
LIN {X 0,Y 186.494,Z 504.143,A -85,B 0,C 180,E1 -22405.678,E2 -22405.678} C_VEL
LIN {X 0,Y 186.483,Z 510.192,A -85,B 0,C 180,E1 -22408.92,E2 -22408.92} C_VEL
LIN {X 0,Y 186.264,Z 513.248,A -85,B 0,C 180,E1 -22411.081,E2 -22411.081} C_VEL
LIN {X 0,Y 185.287,Z 516.618,A -85,B 0,C 180,E1 -22414.351,E2 -22414.351} C_VEL
LIN {X 0,Y 184.564,Z 519.267,A -85,B 0,C 180,E1 -22418.089,E2 -22418.089} C_VEL
LIN {X 0,Y 184.534,Z 520.539,A -85,B 0,C 180,E1 -22420.978,E2 -22420.978} C_VEL
LIN {X 0,Y 185.582,Z 521.453,A -85,B 0,C 180,E1 -22425.373,E2 -22425.373} C_VEL
LIN {X 0,Y 188.044,Z 521.093,A -85,B 0,C 180,E1 -22429.656,E2 -22429.656} C_VEL
LIN {X 0,Y 188.486,Z 520.916,A -85,B 0,C 180,E1 -22430.212,E2 -22430.212} C_VEL
LIN {X 0,Y 189.352,Z 520.306,A -85,B 0,C 180,E1 -22431.977,E2 -22431.977} C_VEL
LIN {X 0,Y 190.025,Z 517.427,A -85,B 0,C 180,E1 -22437.296,E2 -22437.296} C_VEL
LIN {X 0,Y 191.485,Z 516.172,A -85,B 0,C 180,E1 -22438.963,E2 -22438.963} C_VEL
LIN {X 0,Y 192.279,Z 515.687,A -85,B 0,C 180,E1 -22439.479,E2 -22439.479} C_VEL
LIN {X 0,Y 197.441,Z 512.702,A -85,B 0,C 180,E1 -22442.272,E2 -22442.272} C_VEL
LIN {X 0,Y 203.227,Z 508.904,A -85,B 0,C 180,E1 -22444.793,E2 -22444.793} C_VEL
LIN {X 0,Y 209.572,Z 504.287,A -85,B 0,C 180,E1 -22447.131,E2 -22447.131} C_VEL
LIN {X 0,Y 213.637,Z 500.801,A -85,B 0,C 180,E1 -22448.686,E2 -22448.686} C_VEL
LIN {X 0,Y 218.725,Z 495.401,A -85,B 0,C 180,E1 -22451.201,E2 -22451.201} C_VEL
LIN {X 0,Y 219.605,Z 493.866,A -85,B 0,C 180,E1 -22452.227,E2 -22452.227} C_VEL
LIN {X 0,Y 219.651,Z 491.439,A -85,B 0,C 180,E1 -22455.258,E2 -22455.258} C_VEL
LIN {X 0,Y 219.281,Z 490.352,A -85,B 0,C 180,E1 -22457.697,E2 -22457.697} C_VEL
LIN {X 0,Y 218.469,Z 489.994,A -85,B 0,C 180,E1 -22460.54,E2 -22460.54} C_VEL
LIN {X 0,Y 217.902,Z 490.064,A -85,B 0,C 180,E1 -22462.207,E2 -22462.207} C_VEL
LIN {X 0,Y 216.824,Z 490.761,A -85,B 0,C 180,E1 -22464.307,E2 -22464.307} C_VEL
LIN {X 0,Y 215.259,Z 491.863,A -85,B 0,C 180,E1 -22466.287,E2 -22466.287} C_VEL
LIN {X 0,Y 213.387,Z 493.165,A -85,B 0,C 180,E1 -22468.199,E2 -22468.199} C_VEL
LIN {X 0,Y 211.257,Z 494.532,A -85,B 0,C 180,E1 -22470.065,E2 -22470.065} C_VEL
LIN {X 0,Y 207.901,Z 496.224,A -85,B 0,C 180,E1 -22471.754,E2 -22471.754} C_VEL
LIN {X 0,Y 203.895,Z 497.754,A -85,B 0,C 180,E1 -22473.379,E2 -22473.379} C_VEL
LIN {X 0,Y 200.141,Z 498.872,A -85,B 0,C 180,E1 -22475.078,E2 -22475.078} C_VEL
LIN {X 0,Y 196.607,Z 499.478,A -85,B 0,C 180,E1 -22476.846,E2 -22476.846} C_VEL
LIN {X 0,Y 193.319,Z 499.65,A -85,B 0,C 180,E1 -22478.682,E2 -22478.682} C_VEL
LIN {X 0,Y 190.303,Z 499.327,A -85,B 0,C 180,E1 -22480.587,E2 -22480.587} C_VEL
LIN {X 0,Y 187.537,Z 498.546,A -85,B 0,C 180,E1 -22482.554,E2 -22482.554} C_VEL
LIN {X 0,Y 185.03,Z 497.258,A -85,B 0,C 180,E1 -22484.581,E2 -22484.581} C_VEL
LIN {X 0,Y 181.911,Z 494.394,A -85,B 0,C 180,E1 -22487.732,E2 -22487.732} C_VEL
LIN {X 0,Y 179.528,Z 490.341,A -85,B 0,C 180,E1 -22490.991,E2 -22490.991} C_VEL
LIN {X 0,Y 177.989,Z 485.026,A -85,B 0,C 180,E1 -22494.335,E2 -22494.335} C_VEL
LIN {X 0,Y 177.264,Z 478.266,A -85,B 0,C 180,E1 -22497.728,E2 -22497.728} C_VEL
LIN {X 0,Y 177.119,Z 469.806,A -85,B 0,C 180,E1 -22501.137,E2 -22501.137} C_VEL
LIN {X 0,Y 177.588,Z 459.994,A -85,B 0,C 180,E1 -22504.256,E2 -22504.256} C_VEL
LIN {X 0,Y 177.906,Z 449.939,A -85,B 0,C 180,E1 -22506.806,E2 -22506.806} C_VEL
LIN {X 0,Y 178.424,Z 438.885,A -85,B 0,C 180,E1 -22509.065,E2 -22509.065} C_VEL
LIN {X 0,Y 178.464,Z 432.765,A -85,B 0,C 180,E1 -22510.096,E2 -22510.096} C_VEL
LIN {X 0,Y 177.17,Z 420.384,A -85,B 0,C 180,E1 -22511.73,E2 -22511.73} C_VEL
LIN {X 0,Y 177.041,Z 418.93,A -85,B 0,C 180,E1 -22511.957,E2 -22511.957} C_VEL
LIN {X 0,Y 177.189,Z 411.934,A -85,B 0,C 180,E1 -22518.501,E2 -22518.501} C_VEL
LIN {X 0,Y 177.75,Z 406.892,A -85,B 0,C 180,E1 -22523.29,E2 -22523.29} C_VEL
LIN {X 0,Y 178.387,Z 401.782,A -85,B 0,C 180,E1 -22528.215,E2 -22528.215} C_VEL
LIN {X 0,Y 178.937,Z 398.19,A -85,B 0,C 180,E1 -22531.856,E2 -22531.856} C_VEL
LIN {X 0,Y 178.482,Z 398.251,A -85,B 0,C 180,E1 -22538.044,E2 -22538.044} C_VEL
LIN {X 0,Y 178.405,Z 398.258,A -85,B 0,C 180,E1 -22542.044,E2 -22542.044} C_VEL
LIN {X 0,Y 178.398,Z 398.262,A -85,B 0,C 180,E1 -22545.163,E2 -22545.163} C_VEL
LIN {X 0,Y 178.41,Z 398.262,A -85,B 0,C 180,E1 -22548.457,E2 -22548.457} C_VEL
LIN {X 0,Y 178.425,Z 398.257,A -85,B 0,C 180,E1 -22553.783,E2 -22553.783} C_VEL
LIN {X 0,Y 178.488,Z 398.253,A -85,B 0,C 180,E1 -22556.547,E2 -22556.547} C_VEL
LIN {X 0,Y 178.525,Z 398.242,A -85,B 0,C 180,E1 -22560.007,E2 -22560.007} C_VEL
LIN {X 0,Y 178.537,Z 398.245,A -85,B 0,C 180,E1 -22564.876,E2 -22564.876} C_VEL
LIN {X 0,Y 178.641,Z 398.232,A -85,B 0,C 180,E1 -22570.769,E2 -22570.769} C_VEL
LIN {X 0,Y 178.663,Z 398.226,A -85,B 0,C 180,E1 -22576.348,E2 -22576.348} C_VEL
LIN {X 0,Y 178.914,Z 398.197,A -85,B 0,C 180,E1 -22580.96,E2 -22580.96} C_VEL
LIN {X 0,Y 179.156,Z 398.166,A -85,B 0,C 180,E1 -22587.752,E2 -22587.752} C_VEL
LIN {X 0,Y 179.373,Z 398.143,A -85,B 0,C 180,E1 -22590,E2 -22590} C_VEL
LIN {X 0,Y 178.877,Z 398.199,A -85,B 0,C 180,E1 -22594.507,E2 -22594.507} C_VEL
LIN {X 0,Y 178.962,Z 398.191,A -85,B 0,C 180,E1 -22599.038,E2 -22599.038} C_VEL
LIN {X 0,Y 178.691,Z 398.222,A -85,B 0,C 180,E1 -22603.649,E2 -22603.649} C_VEL
LIN {X 0,Y 178.683,Z 398.226,A -85,B 0,C 180,E1 -22608.34,E2 -22608.34} C_VEL
LIN {X 0,Y 178.533,Z 398.243,A -85,B 0,C 180,E1 -22613.182,E2 -22613.182} C_VEL
LIN {X 0,Y 178.49,Z 398.248,A -85,B 0,C 180,E1 -22618.196,E2 -22618.196} C_VEL
LIN {X 0,Y 178.481,Z 398.247,A -85,B 0,C 180,E1 -22620.79,E2 -22620.79} C_VEL
LIN {X 0,Y 178.498,Z 398.249,A -85,B 0,C 180,E1 -22624.225,E2 -22624.225} C_VEL
LIN {X 0,Y 178.419,Z 398.255,A -85,B 0,C 180,E1 -22629.068,E2 -22629.068} C_VEL
LIN {X 0,Y 178.403,Z 398.261,A -85,B 0,C 180,E1 -22632.044,E2 -22632.044} C_VEL
LIN {X 0,Y 178.394,Z 398.263,A -85,B 0,C 180,E1 -22635.164,E2 -22635.164} C_VEL
LIN {X 0,Y 178.404,Z 398.258,A -85,B 0,C 180,E1 -22638.459,E2 -22638.459} C_VEL
LIN {X 0,Y 178.424,Z 398.257,A -85,B 0,C 180,E1 -22643.783,E2 -22643.783} C_VEL
LIN {X 0,Y 178.488,Z 398.247,A -85,B 0,C 180,E1 -22646.547,E2 -22646.547} C_VEL
LIN {X 0,Y 178.524,Z 398.246,A -85,B 0,C 180,E1 -22650.006,E2 -22650.006} C_VEL
LIN {X 0,Y 178.536,Z 398.242,A -85,B 0,C 180,E1 -22654.875,E2 -22654.875} C_VEL
LIN {X 0,Y 178.64,Z 398.232,A -85,B 0,C 180,E1 -22660.769,E2 -22660.769} C_VEL
LIN {X 0,Y 178.677,Z 398.224,A -85,B 0,C 180,E1 -22664.018,E2 -22664.018} C_VEL
LIN {X 0,Y 178.896,Z 398.199,A -85,B 0,C 180,E1 -22669.153,E2 -22669.153} C_VEL
LIN {X 0,Y 178.936,Z 398.194,A -85,B 0,C 180,E1 -22673.233,E2 -22673.233} C_VEL
LIN {X 0,Y 179.156,Z 398.166,A -85,B 0,C 180,E1 -22677.752,E2 -22677.752} C_VEL
LIN {X 0,Y 179.372,Z 398.137,A -85,B 0,C 180,E1 -22680,E2 -22680} C_VEL
LIN {X 0,Y 178.881,Z 398.204,A -85,B 0,C 180,E1 -22684.507,E2 -22684.507} C_VEL
LIN {X 0,Y 178.98,Z 398.186,A -85,B 0,C 180,E1 -22689.037,E2 -22689.037} C_VEL
LIN {X 0,Y 178.689,Z 398.226,A -85,B 0,C 180,E1 -22693.65,E2 -22693.65} C_VEL
LIN {X 0,Y 178.651,Z 398.229,A -85,B 0,C 180,E1 -22698.343,E2 -22698.343} C_VEL
LIN {X 0,Y 178.512,Z 398.247,A -85,B 0,C 180,E1 -22703.185,E2 -22703.185} C_VEL
LIN {X 0,Y 178.487,Z 398.252,A -85,B 0,C 180,E1 -22708.197,E2 -22708.197} C_VEL
LIN {X 0,Y 178.478,Z 398.252,A -85,B 0,C 180,E1 -22710.791,E2 -22710.791} C_VEL
LIN {X 0,Y 178.496,Z 398.247,A -85,B 0,C 180,E1 -22714.224,E2 -22714.224} C_VEL
LIN {X 0,Y 178.421,Z 398.259,A -85,B 0,C 180,E1 -22719.068,E2 -22719.068} C_VEL
LIN {X 0,Y 178.583,Z 398.398,A -85,B 0,C 180,E1 -22724.897,E2 -22724.897} C_VEL
LIN {X 0,Y 179.841,Z 404.563,A -85,B 0,C 180,E1 -22729.643,E2 -22729.643} C_VEL
LIN {X 0,Y 181.333,Z 411.111,A -85,B 0,C 180,E1 -22734.479,E2 -22734.479} C_VEL
LIN {X 0,Y 182.401,Z 415.947,A -85,B 0,C 180,E1 -22737.959,E2 -22737.959} C_VEL
LIN {X 0,Y 181.132,Z 420.282,A -85,B 0,C 180,E1 -22740.987,E2 -22740.987} C_VEL
LIN {X 0,Y 178.607,Z 430.136,A -85,B 0,C 180,E1 -22748.049,E2 -22748.049} C_VEL
LIN {X 0,Y 178.266,Z 434.414,A -85,B 0,C 180,E1 -22751.161,E2 -22751.161} C_VEL
LIN {X 0,Y 178.501,Z 447.686,A -85,B 0,C 180,E1 -22752.53,E2 -22752.53} C_VEL
LIN {X 0,Y 179.317,Z 459.014,A -85,B 0,C 180,E1 -22754.077,E2 -22754.077} C_VEL
LIN {X 0,Y 180.269,Z 469.548,A -85,B 0,C 180,E1 -22755.897,E2 -22755.897} C_VEL
LIN {X 0,Y 179.781,Z 479.037,A -85,B 0,C 180,E1 -22758.069,E2 -22758.069} C_VEL
LIN {X 0,Y 179.535,Z 487.679,A -85,B 0,C 180,E1 -22760.477,E2 -22760.477} C_VEL
LIN {X 0,Y 179.44,Z 495.728,A -85,B 0,C 180,E1 -22763.252,E2 -22763.252} C_VEL
LIN {X 0,Y 179.744,Z 502.405,A -85,B 0,C 180,E1 -22766.077,E2 -22766.077} C_VEL
LIN {X 0,Y 179.73,Z 507.621,A -85,B 0,C 180,E1 -22768.88,E2 -22768.88} C_VEL
LIN {X 0,Y 179.538,Z 510.962,A -85,B 0,C 180,E1 -22771.122,E2 -22771.122} C_VEL
LIN {X 0,Y 178.833,Z 513.515,A -85,B 0,C 180,E1 -22773.38,E2 -22773.38} C_VEL
LIN {X 0,Y 177.948,Z 516.427,A -85,B 0,C 180,E1 -22776.805,E2 -22776.805} C_VEL
LIN {X 0,Y 177.679,Z 518.963,A -85,B 0,C 180,E1 -22781.407,E2 -22781.407} C_VEL
LIN {X 0,Y 178.79,Z 520.211,A -85,B 0,C 180,E1 -22785.972,E2 -22785.972} C_VEL
LIN {X 0,Y 181.653,Z 520.135,A -85,B 0,C 180,E1 -22790.725,E2 -22790.725} C_VEL
LIN {X 0,Y 185.409,Z 518.975,A -85,B 0,C 180,E1 -22794.643,E2 -22794.643} C_VEL
LIN {X 0,Y 190.789,Z 516.487,A -85,B 0,C 180,E1 -22798.612,E2 -22798.612} C_VEL
LIN {X 0,Y 192.279,Z 515.687,A -85,B 0,C 180,E1 -22799.479,E2 -22799.479} C_VEL
LIN {X 0,Y 193.48,Z 514.775,A -85,B 0,C 180,E1 -22800.578,E2 -22800.578} C_VEL
LIN {X 0,Y 194.629,Z 511.635,A -85,B 0,C 180,E1 -22804.448,E2 -22804.448} C_VEL
LIN {X 0,Y 196.193,Z 510.416,A -85,B 0,C 180,E1 -22805.457,E2 -22805.457} C_VEL
LIN {X 0,Y 204.024,Z 505.457,A -85,B 0,C 180,E1 -22808.32,E2 -22808.32} C_VEL
LIN {X 0,Y 208.283,Z 502.315,A -85,B 0,C 180,E1 -22809.875,E2 -22809.875} C_VEL
LIN {X 0,Y 213.021,Z 497.905,A -85,B 0,C 180,E1 -22812.164,E2 -22812.164} C_VEL
LIN {X 0,Y 213.523,Z 497.009,A -85,B 0,C 180,E1 -22812.927,E2 -22812.927} C_VEL
LIN {X 0,Y 213.495,Z 494.76,A -85,B 0,C 180,E1 -22816.404,E2 -22816.404} C_VEL
LIN {X 0,Y 212.776,Z 493.882,A -85,B 0,C 180,E1 -22819.437,E2 -22819.437} C_VEL
LIN {X 0,Y 212.264,Z 493.797,A -85,B 0,C 180,E1 -22821.017,E2 -22821.017} C_VEL
LIN {X 0,Y 211.212,Z 494.059,A -85,B 0,C 180,E1 -22823.206,E2 -22823.206} C_VEL
LIN {X 0,Y 209.633,Z 494.81,A -85,B 0,C 180,E1 -22825.255,E2 -22825.255} C_VEL
LIN {X 0,Y 207.664,Z 495.829,A -85,B 0,C 180,E1 -22827.215,E2 -22827.215} C_VEL
LIN {X 0,Y 205.408,Z 496.89,A -85,B 0,C 180,E1 -22829.121,E2 -22829.121} C_VEL
LIN {X 0,Y 201.841,Z 498.313,A -85,B 0,C 180,E1 -22830.825,E2 -22830.825} C_VEL
LIN {X 0,Y 197.725,Z 499.547,A -85,B 0,C 180,E1 -22832.479,E2 -22832.479} C_VEL
LIN {X 0,Y 193.837,Z 500.331,A -85,B 0,C 180,E1 -22834.209,E2 -22834.209} C_VEL
LIN {X 0,Y 190.183,Z 500.664,A -85,B 0,C 180,E1 -22836.015,E2 -22836.015} C_VEL
LIN {X 0,Y 186.771,Z 500.558,A -85,B 0,C 180,E1 -22837.896,E2 -22837.896} C_VEL
LIN {X 0,Y 183.638,Z 499.955,A -85,B 0,C 180,E1 -22839.853,E2 -22839.853} C_VEL
LIN {X 0,Y 180.77,Z 498.905,A -85,B 0,C 180,E1 -22841.879,E2 -22841.879} C_VEL
LIN {X 0,Y 177.036,Z 496.378,A -85,B 0,C 180,E1 -22845.046,E2 -22845.046} C_VEL
LIN {X 0,Y 174.051,Z 492.749,A -85,B 0,C 180,E1 -22848.352,E2 -22848.352} C_VEL
LIN {X 0,Y 171.961,Z 487.879,A -85,B 0,C 180,E1 -22851.776,E2 -22851.776} C_VEL
LIN {X 0,Y 170.672,Z 481.746,A -85,B 0,C 180,E1 -22855.276,E2 -22855.276} C_VEL
LIN {X 0,Y 170.176,Z 473.949,A -85,B 0,C 180,E1 -22858.817,E2 -22858.817} C_VEL
LIN {X 0,Y 170.326,Z 464.243,A -85,B 0,C 180,E1 -22862.365,E2 -22862.365} C_VEL
LIN {X 0,Y 170.763,Z 455.247,A -85,B 0,C 180,E1 -22865.018,E2 -22865.018} C_VEL
LIN {X 0,Y 171.211,Z 443.891,A -85,B 0,C 180,E1 -22867.667,E2 -22867.667} C_VEL
LIN {X 0,Y 171.532,Z 433.549,A -85,B 0,C 180,E1 -22869.591,E2 -22869.591} C_VEL
LIN {X 0,Y 170.146,Z 420.399,A -85,B 0,C 180,E1 -22871.395,E2 -22871.395} C_VEL
LIN {X 0,Y 170.063,Z 419.366,A -85,B 0,C 180,E1 -22871.531,E2 -22871.531} C_VEL
LIN {X 0,Y 170.162,Z 411.372,A -85,B 0,C 180,E1 -22879.294,E2 -22879.294} C_VEL
LIN {X 0,Y 170.758,Z 406.292,A -85,B 0,C 180,E1 -22884.304,E2 -22884.304} C_VEL
LIN {X 0,Y 171.5,Z 401.128,A -85,B 0,C 180,E1 -22889.456,E2 -22889.456} C_VEL
LIN {X 0,Y 171.884,Z 399.07,A -85,B 0,C 180,E1 -22891.71,E2 -22891.71} C_VEL
LIN {X 0,Y 171.435,Z 399.129,A -85,B 0,C 180,E1 -22897.947,E2 -22897.947} C_VEL
LIN {X 0,Y 171.341,Z 399.138,A -85,B 0,C 180,E1 -22902.411,E2 -22902.411} C_VEL
LIN {X 0,Y 171.345,Z 399.14,A -85,B 0,C 180,E1 -22907.587,E2 -22907.587} C_VEL
LIN {X 0,Y 171.389,Z 399.13,A -85,B 0,C 180,E1 -22912.041,E2 -22912.041} C_VEL
LIN {X 0,Y 171.4,Z 399.134,A -85,B 0,C 180,E1 -22915.092,E2 -22915.092} C_VEL
LIN {X 0,Y 171.451,Z 399.124,A -85,B 0,C 180,E1 -22920.534,E2 -22920.534} C_VEL
LIN {X 0,Y 171.461,Z 399.126,A -85,B 0,C 180,E1 -22925.802,E2 -22925.802} C_VEL
LIN {X 0,Y 171.598,Z 399.109,A -85,B 0,C 180,E1 -22930.874,E2 -22930.874} C_VEL
LIN {X 0,Y 171.583,Z 399.11,A -85,B 0,C 180,E1 -22935.773,E2 -22935.773} C_VEL
LIN {X 0,Y 171.851,Z 399.078,A -85,B 0,C 180,E1 -22940.585,E2 -22940.585} C_VEL
LIN {X 0,Y 171.819,Z 399.077,A -85,B 0,C 180,E1 -22945.307,E2 -22945.307} C_VEL
LIN {X 0,Y 172.336,Z 399.02,A -85,B 0,C 180,E1 -22950,E2 -22950} C_VEL
LIN {X 0,Y 171.825,Z 399.076,A -85,B 0,C 180,E1 -22954.692,E2 -22954.692} C_VEL
LIN {X 0,Y 171.891,Z 399.073,A -85,B 0,C 180,E1 -22959.413,E2 -22959.413} C_VEL
LIN {X 0,Y 171.616,Z 399.106,A -85,B 0,C 180,E1 -22964.224,E2 -22964.224} C_VEL
LIN {X 0,Y 171.578,Z 399.111,A -85,B 0,C 180,E1 -22969.591,E2 -22969.591} C_VEL
LIN {X 0,Y 171.472,Z 399.127,A -85,B 0,C 180,E1 -22975.617,E2 -22975.617} C_VEL
LIN {X 0,Y 171.444,Z 399.124,A -85,B 0,C 180,E1 -22980.587,E2 -22980.587} C_VEL
LIN {X 0,Y 171.409,Z 399.134,A -85,B 0,C 180,E1 -22985.031,E2 -22985.031} C_VEL
LIN {X 0,Y 171.381,Z 399.131,A -85,B 0,C 180,E1 -22988.816,E2 -22988.816} C_VEL
LIN {X 0,Y 171.322,Z 399.142,A -85,B 0,C 180,E1 -22994.217,E2 -22994.217} C_VEL
LIN {X 0,Y 171.336,Z 399.14,A -85,B 0,C 180,E1 -22998.981,E2 -22998.981} C_VEL
LIN {X 0,Y 171.388,Z 399.135,A -85,B 0,C 180,E1 -23002.041,E2 -23002.041} C_VEL
LIN {X 0,Y 171.399,Z 399.131,A -85,B 0,C 180,E1 -23005.092,E2 -23005.092} C_VEL
LIN {X 0,Y 171.451,Z 399.128,A -85,B 0,C 180,E1 -23010.534,E2 -23010.534} C_VEL
LIN {X 0,Y 171.46,Z 399.124,A -85,B 0,C 180,E1 -23015.802,E2 -23015.802} C_VEL
LIN {X 0,Y 171.597,Z 399.108,A -85,B 0,C 180,E1 -23020.873,E2 -23020.873} C_VEL
LIN {X 0,Y 171.615,Z 399.106,A -85,B 0,C 180,E1 -23025.776,E2 -23025.776} C_VEL
LIN {X 0,Y 171.912,Z 399.067,A -85,B 0,C 180,E1 -23030.588,E2 -23030.588} C_VEL
LIN {X 0,Y 171.827,Z 399.08,A -85,B 0,C 180,E1 -23035.308,E2 -23035.308} C_VEL
LIN {X 0,Y 172.335,Z 399.013,A -85,B 0,C 180,E1 -23040,E2 -23040} C_VEL
LIN {X 0,Y 171.83,Z 399.081,A -85,B 0,C 180,E1 -23044.692,E2 -23044.692} C_VEL
LIN {X 0,Y 171.912,Z 399.066,A -85,B 0,C 180,E1 -23049.411,E2 -23049.411} C_VEL
LIN {X 0,Y 171.611,Z 399.109,A -85,B 0,C 180,E1 -23054.224,E2 -23054.224} C_VEL
LIN {X 0,Y 171.546,Z 399.114,A -85,B 0,C 180,E1 -23059.562,E2 -23059.562} C_VEL
LIN {X 0,Y 171.47,Z 399.122,A -85,B 0,C 180,E1 -23065.616,E2 -23065.616} C_VEL
LIN {X 0,Y 171.44,Z 399.129,A -85,B 0,C 180,E1 -23070.585,E2 -23070.585} C_VEL
LIN {X 0,Y 171.406,Z 399.129,A -85,B 0,C 180,E1 -23075.032,E2 -23075.032} C_VEL
LIN {X 0,Y 171.382,Z 399.136,A -85,B 0,C 180,E1 -23078.817,E2 -23078.817} C_VEL
LIN {X 0,Y 171.545,Z 399.288,A -85,B 0,C 180,E1 -23084.846,E2 -23084.846} C_VEL
LIN {X 0,Y 173.031,Z 406.381,A -85,B 0,C 180,E1 -23090.509,E2 -23090.509} C_VEL
LIN {X 0,Y 174.954,Z 414.375,A -85,B 0,C 180,E1 -23096.63,E2 -23096.63} C_VEL
LIN {X 0,Y 175.248,Z 415.357,A -85,B 0,C 180,E1 -23097.37,E2 -23097.37} C_VEL
LIN {X 0,Y 175.114,Z 416.971,A -85,B 0,C 180,E1 -23098.551,E2 -23098.551} C_VEL
LIN {X 0,Y 172.525,Z 425.219,A -85,B 0,C 180,E1 -23104.676,E2 -23104.676} C_VEL
LIN {X 0,Y 171.246,Z 434.081,A -85,B 0,C 180,E1 -23111.454,E2 -23111.454} C_VEL
LIN {X 0,Y 171.501,Z 447.201,A -85,B 0,C 180,E1 -23112.87,E2 -23112.87} C_VEL
LIN {X 0,Y 172.421,Z 459.44,A -85,B 0,C 180,E1 -23114.636,E2 -23114.636} C_VEL
LIN {X 0,Y 173.327,Z 468.176,A -85,B 0,C 180,E1 -23116.211,E2 -23116.211} C_VEL
LIN {X 0,Y 172.921,Z 478.064,A -85,B 0,C 180,E1 -23118.572,E2 -23118.572} C_VEL
LIN {X 0,Y 172.718,Z 487.087,A -85,B 0,C 180,E1 -23121.223,E2 -23121.223} C_VEL
LIN {X 0,Y 172.721,Z 495.161,A -85,B 0,C 180,E1 -23124.162,E2 -23124.162} C_VEL
LIN {X 0,Y 173.032,Z 501.736,A -85,B 0,C 180,E1 -23127.09,E2 -23127.09} C_VEL
LIN {X 0,Y 172.976,Z 506.841,A -85,B 0,C 180,E1 -23130,E2 -23130} C_VEL
LIN {X 0,Y 172.561,Z 509.999,A -85,B 0,C 180,E1 -23132.334,E2 -23132.334} C_VEL
LIN {X 0,Y 171.178,Z 514.382,A -85,B 0,C 180,E1 -23137.075,E2 -23137.075} C_VEL
LIN {X 0,Y 170.874,Z 517.261,A -85,B 0,C 180,E1 -23141.868,E2 -23141.868} C_VEL
LIN {X 0,Y 172.053,Z 518.821,A -85,B 0,C 180,E1 -23146.615,E2 -23146.615} C_VEL
LIN {X 0,Y 174.789,Z 519.184,A -85,B 0,C 180,E1 -23151.216,E2 -23151.216} C_VEL
LIN {X 0,Y 178.992,Z 518.375,A -85,B 0,C 180,E1 -23155.589,E2 -23155.589} C_VEL
LIN {X 0,Y 184.586,Z 516.321,A -85,B 0,C 180,E1 -23159.668,E2 -23159.668} C_VEL
LIN {X 0,Y 191.497,Z 513.015,A -85,B 0,C 180,E1 -23163.402,E2 -23163.402} C_VEL
LIN {X 0,Y 196.193,Z 510.416,A -85,B 0,C 180,E1 -23165.457,E2 -23165.457} C_VEL
LIN {X 0,Y 197.889,Z 509.172,A -85,B 0,C 180,E1 -23166.436,E2 -23166.436} C_VEL
LIN {X 0,Y 199.315,Z 507.312,A -85,B 0,C 180,E1 -23168.253,E2 -23168.253} C_VEL
LIN {X 0,Y 200.812,Z 505.345,A -85,B 0,C 180,E1 -23170.054,E2 -23170.054} C_VEL
LIN {X 0,Y 202.585,Z 503.928,A -85,B 0,C 180,E1 -23170.991,E2 -23170.991} C_VEL
LIN {X 0,Y 206.746,Z 500.714,A -85,B 0,C 180,E1 -23172.834,E2 -23172.834} C_VEL
LIN {X 0,Y 207.27,Z 499.287,A -85,B 0,C 180,E1 -23174.598,E2 -23174.598} C_VEL
LIN {X 0,Y 207.1,Z 497.953,A -85,B 0,C 180,E1 -23177.257,E2 -23177.257} C_VEL
LIN {X 0,Y 206.465,Z 497.333,A -85,B 0,C 180,E1 -23179.703,E2 -23179.703} C_VEL
LIN {X 0,Y 205.448,Z 497.233,A -85,B 0,C 180,E1 -23181.994,E2 -23181.994} C_VEL
LIN {X 0,Y 203.94,Z 497.631,A -85,B 0,C 180,E1 -23184.138,E2 -23184.138} C_VEL
LIN {X 0,Y 200.741,Z 498.737,A -85,B 0,C 180,E1 -23187.167,E2 -23187.167} C_VEL
LIN {X 0,Y 199.569,Z 499.116,A -85,B 0,C 180,E1 -23188.114,E2 -23188.114} C_VEL
LIN {X 0,Y 195.804,Z 500.228,A -85,B 0,C 180,E1 -23189.834,E2 -23189.834} C_VEL
LIN {X 0,Y 191.559,Z 501.16,A -85,B 0,C 180,E1 -23191.514,E2 -23191.514} C_VEL
LIN {X 0,Y 187.546,Z 501.653,A -85,B 0,C 180,E1 -23193.277,E2 -23193.277} C_VEL
LIN {X 0,Y 183.763,Z 501.689,A -85,B 0,C 180,E1 -23195.122,E2 -23195.122} C_VEL
LIN {X 0,Y 180.243,Z 501.289,A -85,B 0,C 180,E1 -23197.051,E2 -23197.051} C_VEL
LIN {X 0,Y 176.986,Z 500.413,A -85,B 0,C 180,E1 -23199.06,E2 -23199.06} C_VEL
LIN {X 0,Y 174.027,Z 499.084,A -85,B 0,C 180,E1 -23201.151,E2 -23201.151} C_VEL
LIN {X 0,Y 170.189,Z 496.164,A -85,B 0,C 180,E1 -23204.43,E2 -23204.43} C_VEL
LIN {X 0,Y 167.131,Z 492.121,A -85,B 0,C 180,E1 -23207.863,E2 -23207.863} C_VEL
LIN {X 0,Y 164.99,Z 486.873,A -85,B 0,C 180,E1 -23211.426,E2 -23211.426} C_VEL
LIN {X 0,Y 163.713,Z 480.256,A -85,B 0,C 180,E1 -23215.075,E2 -23215.075} C_VEL
LIN {X 0,Y 163.255,Z 472.068,A -85,B 0,C 180,E1 -23218.767,E2 -23218.767} C_VEL
LIN {X 0,Y 163.479,Z 461.71,A -85,B 0,C 180,E1 -23222.464,E2 -23222.464} C_VEL
LIN {X 0,Y 163.848,Z 453.267,A -85,B 0,C 180,E1 -23224.922,E2 -23224.922} C_VEL
LIN {X 0,Y 164.246,Z 441.485,A -85,B 0,C 180,E1 -23227.685,E2 -23227.685} C_VEL
LIN {X 0,Y 164.539,Z 433.266,A -85,B 0,C 180,E1 -23229.217,E2 -23229.217} C_VEL
LIN {X 0,Y 163.065,Z 419.655,A -85,B 0,C 180,E1 -23231.183,E2 -23231.183} C_VEL
LIN {X 0,Y 163.182,Z 410.771,A -85,B 0,C 180,E1 -23240.154,E2 -23240.154} C_VEL
LIN {X 0,Y 163.845,Z 405.328,A -85,B 0,C 180,E1 -23245.739,E2 -23245.739} C_VEL
LIN {X 0,Y 164.802,Z 399.956,A -85,B 0,C 180,E1 -23251.47,E2 -23251.47} C_VEL
LIN {X 0,Y 164.4,Z 400.005,A -85,B 0,C 180,E1 -23256.762,E2 -23256.762} C_VEL
LIN {X 0,Y 164.309,Z 400.016,A -85,B 0,C 180,E1 -23259.912,E2 -23259.912} C_VEL
LIN {X 0,Y 164.281,Z 400.017,A -85,B 0,C 180,E1 -23263.342,E2 -23263.342} C_VEL
LIN {X 0,Y 164.294,Z 400.021,A -85,B 0,C 180,E1 -23266.809,E2 -23266.809} C_VEL
LIN {X 0,Y 164.298,Z 400.017,A -85,B 0,C 180,E1 -23270.352,E2 -23270.352} C_VEL
LIN {X 0,Y 164.332,Z 400.014,A -85,B 0,C 180,E1 -23274.349,E2 -23274.349} C_VEL
LIN {X 0,Y 164.392,Z 400.002,A -85,B 0,C 180,E1 -23279.135,E2 -23279.135} C_VEL
LIN {X 0,Y 164.419,Z 400.004,A -85,B 0,C 180,E1 -23284.694,E2 -23284.694} C_VEL
LIN {X 0,Y 164.489,Z 399.992,A -85,B 0,C 180,E1 -23290.05,E2 -23290.05} C_VEL
LIN {X 0,Y 164.533,Z 399.987,A -85,B 0,C 180,E1 -23295.15,E2 -23295.15} C_VEL
LIN {X 0,Y 164.771,Z 399.961,A -85,B 0,C 180,E1 -23300.176,E2 -23300.176} C_VEL
LIN {X 0,Y 164.834,Z 399.951,A -85,B 0,C 180,E1 -23302.651,E2 -23302.651} C_VEL
LIN {X 0,Y 165.051,Z 399.922,A -85,B 0,C 180,E1 -23307.559,E2 -23307.559} C_VEL
LIN {X 0,Y 165.298,Z 399.896,A -85,B 0,C 180,E1 -23310,E2 -23310} C_VEL
LIN {X 0,Y 164.775,Z 399.954,A -85,B 0,C 180,E1 -23314.893,E2 -23314.893} C_VEL
LIN {X 0,Y 164.854,Z 399.949,A -85,B 0,C 180,E1 -23317.348,E2 -23317.348} C_VEL
LIN {X 0,Y 164.756,Z 399.96,A -85,B 0,C 180,E1 -23321.152,E2 -23321.152} C_VEL
LIN {X 0,Y 164.529,Z 399.991,A -85,B 0,C 180,E1 -23327.398,E2 -23327.398} C_VEL
LIN {X 0,Y 164.522,Z 399.988,A -85,B 0,C 180,E1 -23329.983,E2 -23329.983} C_VEL
LIN {X 0,Y 164.396,Z 400.006,A -85,B 0,C 180,E1 -23336.134,E2 -23336.134} C_VEL
LIN {X 0,Y 164.378,Z 400.005,A -85,B 0,C 180,E1 -23341.228,E2 -23341.228} C_VEL
LIN {X 0,Y 164.315,Z 400.015,A -85,B 0,C 180,E1 -23346.784,E2 -23346.784} C_VEL
LIN {X 0,Y 164.301,Z 400.016,A -85,B 0,C 180,E1 -23349.913,E2 -23349.913} C_VEL
LIN {X 0,Y 164.28,Z 400.022,A -85,B 0,C 180,E1 -23353.342,E2 -23353.342} C_VEL
LIN {X 0,Y 164.264,Z 400.019,A -85,B 0,C 180,E1 -23356.799,E2 -23356.799} C_VEL
LIN {X 0,Y 164.296,Z 400.018,A -85,B 0,C 180,E1 -23360.352,E2 -23360.352} C_VEL
LIN {X 0,Y 164.331,Z 400.009,A -85,B 0,C 180,E1 -23366.222,E2 -23366.222} C_VEL
LIN {X 0,Y 164.407,Z 400.007,A -85,B 0,C 180,E1 -23369.138,E2 -23369.138} C_VEL
LIN {X 0,Y 164.418,Z 399.999,A -85,B 0,C 180,E1 -23374.694,E2 -23374.694} C_VEL
LIN {X 0,Y 164.487,Z 399.994,A -85,B 0,C 180,E1 -23380.049,E2 -23380.049} C_VEL
LIN {X 0,Y 164.561,Z 399.986,A -85,B 0,C 180,E1 -23385.152,E2 -23385.152} C_VEL
LIN {X 0,Y 164.855,Z 399.948,A -85,B 0,C 180,E1 -23390.181,E2 -23390.181} C_VEL
LIN {X 0,Y 164.864,Z 399.945,A -85,B 0,C 180,E1 -23392.652,E2 -23392.652} C_VEL
LIN {X 0,Y 165.053,Z 399.923,A -85,B 0,C 180,E1 -23397.559,E2 -23397.559} C_VEL
LIN {X 0,Y 165.298,Z 399.89,A -85,B 0,C 180,E1 -23400,E2 -23400} C_VEL
LIN {X 0,Y 164.78,Z 399.959,A -85,B 0,C 180,E1 -23404.893,E2 -23404.893} C_VEL
LIN {X 0,Y 164.854,Z 399.946,A -85,B 0,C 180,E1 -23409.818,E2 -23409.818} C_VEL
LIN {X 0,Y 164.555,Z 399.985,A -85,B 0,C 180,E1 -23414.848,E2 -23414.848} C_VEL
LIN {X 0,Y 164.474,Z 399.997,A -85,B 0,C 180,E1 -23419.989,E2 -23419.989} C_VEL
LIN {X 0,Y 164.394,Z 400.003,A -85,B 0,C 180,E1 -23426.134,E2 -23426.134} C_VEL
LIN {X 0,Y 164.375,Z 400.008,A -85,B 0,C 180,E1 -23431.227,E2 -23431.227} C_VEL
LIN {X 0,Y 164.314,Z 400.015,A -85,B 0,C 180,E1 -23436.784,E2 -23436.784} C_VEL
LIN {X 0,Y 164.303,Z 400.018,A -85,B 0,C 180,E1 -23439.913,E2 -23439.913} C_VEL
LIN {X 0,Y 164.485,Z 400.175,A -85,B 0,C 180,E1 -23444.836,E2 -23444.836} C_VEL
LIN {X 0,Y 165.73,Z 406.057,A -85,B 0,C 180,E1 -23449.757,E2 -23449.757} C_VEL
LIN {X 0,Y 167.458,Z 413.155,A -85,B 0,C 180,E1 -23455.471,E2 -23455.471} C_VEL
LIN {X 0,Y 167.997,Z 415.153,A -85,B 0,C 180,E1 -23457.055,E2 -23457.055} C_VEL
LIN {X 0,Y 167.971,Z 416.981,A -85,B 0,C 180,E1 -23458.466,E2 -23458.466} C_VEL
LIN {X 0,Y 165.356,Z 425.126,A -85,B 0,C 180,E1 -23464.848,E2 -23464.848} C_VEL
LIN {X 0,Y 164.248,Z 433.782,A -85,B 0,C 180,E1 -23471.835,E2 -23471.835} C_VEL
LIN {X 0,Y 164.572,Z 447.272,A -85,B 0,C 180,E1 -23473.406,E2 -23473.406} C_VEL
LIN {X 0,Y 165.567,Z 459.34,A -85,B 0,C 180,E1 -23475.245,E2 -23475.245} C_VEL
LIN {X 0,Y 166.422,Z 466.863,A -85,B 0,C 180,E1 -23476.656,E2 -23476.656} C_VEL
LIN {X 0,Y 166.146,Z 475.431,A -85,B 0,C 180,E1 -23478.718,E2 -23478.718} C_VEL
LIN {X 0,Y 165.98,Z 484.771,A -85,B 0,C 180,E1 -23481.478,E2 -23481.478} C_VEL
LIN {X 0,Y 166.005,Z 493.133,A -85,B 0,C 180,E1 -23484.534,E2 -23484.534} C_VEL
LIN {X 0,Y 166.334,Z 499.878,A -85,B 0,C 180,E1 -23487.579,E2 -23487.579} C_VEL
LIN {X 0,Y 166.313,Z 504.08,A -85,B 0,C 180,E1 -23490,E2 -23490} C_VEL
LIN {X 0,Y 165.945,Z 507.469,A -85,B 0,C 180,E1 -23492.427,E2 -23492.427} C_VEL
LIN {X 0,Y 164.438,Z 512.229,A -85,B 0,C 180,E1 -23497.367,E2 -23497.367} C_VEL
LIN {X 0,Y 164.132,Z 515.395,A -85,B 0,C 180,E1 -23502.363,E2 -23502.363} C_VEL
LIN {X 0,Y 165.384,Z 517.294,A -85,B 0,C 180,E1 -23507.306,E2 -23507.306} C_VEL
LIN {X 0,Y 168.253,Z 518.032,A -85,B 0,C 180,E1 -23512.082,E2 -23512.082} C_VEL
LIN {X 0,Y 172.629,Z 517.619,A -85,B 0,C 180,E1 -23516.605,E2 -23516.605} C_VEL
LIN {X 0,Y 178.459,Z 516.002,A -85,B 0,C 180,E1 -23520.795,E2 -23520.795} C_VEL
LIN {X 0,Y 185.614,Z 513.21,A -85,B 0,C 180,E1 -23524.608,E2 -23524.608} C_VEL
LIN {X 0,Y 193.993,Z 509.083,A -85,B 0,C 180,E1 -23528.016,E2 -23528.016} C_VEL
LIN {X 0,Y 200.839,Z 505.111,A -85,B 0,C 180,E1 -23530.344,E2 -23530.344} C_VEL
LIN {X 0,Y 202.585,Z 503.928,A -85,B 0,C 180,E1 -23530.991,E2 -23530.991} C_VEL
LIN {X 0,Y 203.714,Z 502.918,A -85,B 0,C 180,E1 -23531.764,E2 -23531.764} C_VEL
LIN {X 0,Y 203.771,Z 502.171,A -85,B 0,C 180,E1 -23532.836,E2 -23532.836} C_VEL
LIN {X 0,Y 203.157,Z 501.848,A -85,B 0,C 180,E1 -23533.749,E2 -23533.749} C_VEL
LIN {X 0,Y 200.788,Z 501.305,A -85,B 0,C 180,E1 -23536.559,E2 -23536.559} C_VEL
LIN {X 0,Y 200.706,Z 501.149,A -85,B 0,C 180,E1 -23536.97,E2 -23536.97} C_VEL
LIN {X 0,Y 200.478,Z 500.697,A -85,B 0,C 180,E1 -23538.236,E2 -23538.236} C_VEL
LIN {X 0,Y 199.463,Z 500.278,A -85,B 0,C 180,E1 -23540.82,E2 -23540.82} C_VEL
LIN {X 0,Y 198.121,Z 500.278,A -85,B 0,C 180,E1 -23542.912,E2 -23542.912} C_VEL
LIN {X 0,Y 195.087,Z 500.872,A -85,B 0,C 180,E1 -23545.953,E2 -23545.953} C_VEL
LIN {X 0,Y 193.74,Z 501.141,A -85,B 0,C 180,E1 -23547.035,E2 -23547.035} C_VEL
LIN {X 0,Y 189.809,Z 501.987,A -85,B 0,C 180,E1 -23548.777,E2 -23548.777} C_VEL
LIN {X 0,Y 185.425,Z 502.596,A -85,B 0,C 180,E1 -23550.48,E2 -23550.48} C_VEL
LIN {X 0,Y 181.286,Z 502.787,A -85,B 0,C 180,E1 -23552.276,E2 -23552.276} C_VEL
LIN {X 0,Y 177.367,Z 502.543,A -85,B 0,C 180,E1 -23554.16,E2 -23554.16} C_VEL
LIN {X 0,Y 173.74,Z 501.844,A -85,B 0,C 180,E1 -23556.139,E2 -23556.139} C_VEL
LIN {X 0,Y 170.36,Z 500.695,A -85,B 0,C 180,E1 -23558.205,E2 -23558.205} C_VEL
LIN {X 0,Y 165.924,Z 498.083,A -85,B 0,C 180,E1 -23561.478,E2 -23561.478} C_VEL
LIN {X 0,Y 162.265,Z 494.425,A -85,B 0,C 180,E1 -23564.938,E2 -23564.938} C_VEL
LIN {X 0,Y 159.431,Z 489.551,A -85,B 0,C 180,E1 -23568.559,E2 -23568.559} C_VEL
LIN {X 0,Y 157.499,Z 483.488,A -85,B 0,C 180,E1 -23572.307,E2 -23572.307} C_VEL
LIN {X 0,Y 156.59,Z 475.878,A -85,B 0,C 180,E1 -23576.14,E2 -23576.14} C_VEL
LIN {X 0,Y 156.36,Z 466.525,A -85,B 0,C 180,E1 -23580,E2 -23580} C_VEL
LIN {X 0,Y 156.767,Z 456.839,A -85,B 0,C 180,E1 -23583.213,E2 -23583.213} C_VEL
LIN {X 0,Y 157.126,Z 445.888,A -85,B 0,C 180,E1 -23586.098,E2 -23586.098} C_VEL
LIN {X 0,Y 157.574,Z 434.054,A -85,B 0,C 180,E1 -23588.565,E2 -23588.565} C_VEL
LIN {X 0,Y 156.319,Z 422.156,A -85,B 0,C 180,E1 -23590.361,E2 -23590.361} C_VEL
LIN {X 0,Y 156.127,Z 420.006,A -85,B 0,C 180,E1 -23590.701,E2 -23590.701} C_VEL
LIN {X 0,Y 156.05,Z 411.333,A -85,B 0,C 180,E1 -23599.813,E2 -23599.813} C_VEL
LIN {X 0,Y 156.663,Z 406.392,A -85,B 0,C 180,E1 -23605.077,E2 -23605.077} C_VEL
LIN {X 0,Y 157.625,Z 400.852,A -85,B 0,C 180,E1 -23611.088,E2 -23611.088} C_VEL
LIN {X 0,Y 157.418,Z 400.873,A -85,B 0,C 180,E1 -23615.478,E2 -23615.478} C_VEL
LIN {X 0,Y 157.219,Z 400.901,A -85,B 0,C 180,E1 -23620.541,E2 -23620.541} C_VEL
LIN {X 0,Y 157.179,Z 400.904,A -85,B 0,C 180,E1 -23625.677,E2 -23625.677} C_VEL
LIN {X 0,Y 157.208,Z 400.899,A -85,B 0,C 180,E1 -23629.464,E2 -23629.464} C_VEL
LIN {X 0,Y 157.281,Z 400.893,A -85,B 0,C 180,E1 -23634.486,E2 -23634.486} C_VEL
LIN {X 0,Y 157.295,Z 400.89,A -85,B 0,C 180,E1 -23638.096,E2 -23638.096} C_VEL
LIN {X 0,Y 157.325,Z 400.887,A -85,B 0,C 180,E1 -23643.466,E2 -23643.466} C_VEL
LIN {X 0,Y 157.398,Z 400.874,A -85,B 0,C 180,E1 -23649.666,E2 -23649.666} C_VEL
LIN {X 0,Y 157.464,Z 400.869,A -85,B 0,C 180,E1 -23654.467,E2 -23654.467} C_VEL
LIN {X 0,Y 157.692,Z 400.84,A -85,B 0,C 180,E1 -23659.731,E2 -23659.731} C_VEL
LIN {X 0,Y 157.771,Z 400.832,A -85,B 0,C 180,E1 -23662.32,E2 -23662.32} C_VEL
LIN {X 0,Y 158.261,Z 400.773,A -85,B 0,C 180,E1 -23670,E2 -23670} C_VEL
LIN {X 0,Y 157.812,Z 400.827,A -85,B 0,C 180,E1 -23677.678,E2 -23677.678} C_VEL
LIN {X 0,Y 157.686,Z 400.841,A -85,B 0,C 180,E1 -23681.322,E2 -23681.322} C_VEL
LIN {X 0,Y 157.49,Z 400.866,A -85,B 0,C 180,E1 -23685.53,E2 -23685.53} C_VEL
LIN {X 0,Y 157.418,Z 400.871,A -85,B 0,C 180,E1 -23690.926,E2 -23690.926} C_VEL
LIN {X 0,Y 157.317,Z 400.888,A -85,B 0,C 180,E1 -23696.685,E2 -23696.685} C_VEL
LIN {X 0,Y 157.28,Z 400.891,A -85,B 0,C 180,E1 -23702.426,E2 -23702.426} C_VEL
LIN {X 0,Y 157.285,Z 400.89,A -85,B 0,C 180,E1 -23706.457,E2 -23706.457} C_VEL
LIN {X 0,Y 157.214,Z 400.901,A -85,B 0,C 180,E1 -23712.11,E2 -23712.11} C_VEL
LIN {X 0,Y 157.194,Z 400.9,A -85,B 0,C 180,E1 -23717.883,E2 -23717.883} C_VEL
LIN {X 0,Y 157.269,Z 400.892,A -85,B 0,C 180,E1 -23723.55,E2 -23723.55} C_VEL
LIN {X 0,Y 157.302,Z 400.888,A -85,B 0,C 180,E1 -23728.091,E2 -23728.091} C_VEL
LIN {X 0,Y 157.324,Z 400.882,A -85,B 0,C 180,E1 -23733.466,E2 -23733.466} C_VEL
LIN {X 0,Y 157.397,Z 400.877,A -85,B 0,C 180,E1 -23739.665,E2 -23739.665} C_VEL
LIN {X 0,Y 157.487,Z 400.864,A -85,B 0,C 180,E1 -23744.469,E2 -23744.469} C_VEL
LIN {X 0,Y 157.774,Z 400.829,A -85,B 0,C 180,E1 -23749.736,E2 -23749.736} C_VEL
LIN {X 0,Y 157.826,Z 400.82,A -85,B 0,C 180,E1 -23752.323,E2 -23752.323} C_VEL
LIN {X 0,Y 158.26,Z 400.766,A -85,B 0,C 180,E1 -23760,E2 -23760} C_VEL
LIN {X 0,Y 157.826,Z 400.821,A -85,B 0,C 180,E1 -23767.677,E2 -23767.677} C_VEL
LIN {X 0,Y 157.707,Z 400.838,A -85,B 0,C 180,E1 -23771.362,E2 -23771.362} C_VEL
LIN {X 0,Y 157.48,Z 400.866,A -85,B 0,C 180,E1 -23775.531,E2 -23775.531} C_VEL
LIN {X 0,Y 157.371,Z 400.881,A -85,B 0,C 180,E1 -23780.933,E2 -23780.933} C_VEL
LIN {X 0,Y 157.315,Z 400.886,A -85,B 0,C 180,E1 -23786.684,E2 -23786.684} C_VEL
LIN {X 0,Y 157.278,Z 400.891,A -85,B 0,C 180,E1 -23792.427,E2 -23792.427} C_VEL
LIN {X 0,Y 157.283,Z 400.892,A -85,B 0,C 180,E1 -23796.457,E2 -23796.457} C_VEL
LIN {X 0,Y 157.266,Z 400.89,A -85,B 0,C 180,E1 -23802.092,E2 -23802.092} C_VEL
LIN {X 0,Y 157.446,Z 401.074,A -85,B 0,C 180,E1 -23804.879,E2 -23804.879} C_VEL
LIN {X 0,Y 158.83,Z 407.355,A -85,B 0,C 180,E1 -23810.369,E2 -23810.369} C_VEL
LIN {X 0,Y 160.598,Z 414.336,A -85,B 0,C 180,E1 -23816.25,E2 -23816.25} C_VEL
LIN {X 0,Y 160.905,Z 415.697,A -85,B 0,C 180,E1 -23817.362,E2 -23817.362} C_VEL
LIN {X 0,Y 160.828,Z 416.94,A -85,B 0,C 180,E1 -23818.373,E2 -23818.373} C_VEL
LIN {X 0,Y 158.173,Z 424.979,A -85,B 0,C 180,E1 -23825.032,E2 -23825.032} C_VEL
LIN {X 0,Y 157.264,Z 433.464,A -85,B 0,C 180,E1 -23832.275,E2 -23832.275} C_VEL
LIN {X 0,Y 157.671,Z 447.324,A -85,B 0,C 180,E1 -23833.99,E2 -23833.99} C_VEL
LIN {X 0,Y 158.763,Z 459.495,A -85,B 0,C 180,E1 -23835.958,E2 -23835.958} C_VEL
LIN {X 0,Y 159.607,Z 467.662,A -85,B 0,C 180,E1 -23837.605,E2 -23837.605} C_VEL
LIN {X 0,Y 159.286,Z 478.347,A -85,B 0,C 180,E1 -23840.476,E2 -23840.476} C_VEL
LIN {X 0,Y 159.29,Z 487.694,A -85,B 0,C 180,E1 -23843.667,E2 -23843.667} C_VEL
LIN {X 0,Y 159.596,Z 495.233,A -85,B 0,C 180,E1 -23846.845,E2 -23846.845} C_VEL
LIN {X 0,Y 159.736,Z 500.08,A -85,B 0,C 180,E1 -23849.37,E2 -23849.37} C_VEL
LIN {X 0,Y 159.611,Z 503.079,A -85,B 0,C 180,E1 -23851.262,E2 -23851.262} C_VEL
LIN {X 0,Y 159.363,Z 504.797,A -85,B 0,C 180,E1 -23852.528,E2 -23852.528} C_VEL
LIN {X 0,Y 158.051,Z 508.749,A -85,B 0,C 180,E1 -23856.383,E2 -23856.383} C_VEL
LIN {X 0,Y 157.39,Z 512.103,A -85,B 0,C 180,E1 -23860.772,E2 -23860.772} C_VEL
LIN {X 0,Y 157.899,Z 514.634,A -85,B 0,C 180,E1 -23865.489,E2 -23865.489} C_VEL
LIN {X 0,Y 160.079,Z 516.315,A -85,B 0,C 180,E1 -23870.563,E2 -23870.563} C_VEL
LIN {X 0,Y 163.843,Z 516.85,A -85,B 0,C 180,E1 -23875.401,E2 -23875.401} C_VEL
LIN {X 0,Y 169.202,Z 516.26,A -85,B 0,C 180,E1 -23879.897,E2 -23879.897} C_VEL
LIN {X 0,Y 176.04,Z 514.535,A -85,B 0,C 180,E1 -23883.981,E2 -23883.981} C_VEL
LIN {X 0,Y 184.009,Z 511.617,A -85,B 0,C 180,E1 -23887.669,E2 -23887.669} C_VEL
LIN {X 0,Y 193.175,Z 507.375,A -85,B 0,C 180,E1 -23890.91,E2 -23890.91} C_VEL
LIN {X 0,Y 197.749,Z 504.829,A -85,B 0,C 180,E1 -23892.475,E2 -23892.475} C_VEL
LIN {X 0,Y 199.756,Z 503.518,A -85,B 0,C 180,E1 -23893.32,E2 -23893.32} C_VEL
LIN {X 0,Y 200.704,Z 502.443,A -85,B 0,C 180,E1 -23894.454,E2 -23894.454} C_VEL
LIN {X 0,Y 200.836,Z 501.746,A -85,B 0,C 180,E1 -23895.583,E2 -23895.583} C_VEL
LIN {X 0,Y 200.706,Z 501.149,A -85,B 0,C 180,E1 -23896.97,E2 -23896.97} C_VEL
LIN {X 0,Y 200.251,Z 500.877,A -85,B 0,C 180,E1 -23898.078,E2 -23898.078} C_VEL
LIN {X 0,Y 198.443,Z 501.05,A -85,B 0,C 180,E1 -23899.696,E2 -23899.696} C_VEL
LIN {X 0,Y 195.823,Z 501.603,A -85,B 0,C 180,E1 -23901.249,E2 -23901.249} C_VEL
LIN {X 0,Y 189.86,Z 502.792,A -85,B 0,C 180,E1 -23904.462,E2 -23904.462} C_VEL
LIN {X 0,Y 188.233,Z 502.978,A -85,B 0,C 180,E1 -23905.61,E2 -23905.61} C_VEL
LIN {X 0,Y 187.913,Z 503.003,A -85,B 0,C 180,E1 -23905.875,E2 -23905.875} C_VEL
LIN {X 0,Y 183.85,Z 503.539,A -85,B 0,C 180,E1 -23907.644,E2 -23907.644} C_VEL
LIN {X 0,Y 179.347,Z 503.851,A -85,B 0,C 180,E1 -23909.375,E2 -23909.375} C_VEL
LIN {X 0,Y 175.064,Z 503.737,A -85,B 0,C 180,E1 -23911.201,E2 -23911.201} C_VEL
LIN {X 0,Y 171.029,Z 503.202,A -85,B 0,C 180,E1 -23913.127,E2 -23913.127} C_VEL
LIN {X 0,Y 167.261,Z 502.204,A -85,B 0,C 180,E1 -23915.154,E2 -23915.154} C_VEL
LIN {X 0,Y 163.769,Z 500.779,A -85,B 0,C 180,E1 -23917.28,E2 -23917.28} C_VEL
LIN {X 0,Y 159.214,Z 497.75,A -85,B 0,C 180,E1 -23920.667,E2 -23920.667} C_VEL
LIN {X 0,Y 155.447,Z 493.668,A -85,B 0,C 180,E1 -23924.26,E2 -23924.26} C_VEL
LIN {X 0,Y 152.559,Z 488.401,A -85,B 0,C 180,E1 -23928.036,E2 -23928.036} C_VEL
LIN {X 0,Y 150.6,Z 481.847,A -85,B 0,C 180,E1 -23931.952,E2 -23931.952} C_VEL
LIN {X 0,Y 149.699,Z 473.827,A -85,B 0,C 180,E1 -23935.962,E2 -23935.962} C_VEL
LIN {X 0,Y 149.574,Z 463.83,A -85,B 0,C 180,E1 -23940,E2 -23940} C_VEL
LIN {X 0,Y 150.011,Z 453.599,A -85,B 0,C 180,E1 -23943.358,E2 -23943.358} C_VEL
LIN {X 0,Y 150.337,Z 441.709,A -85,B 0,C 180,E1 -23946.375,E2 -23946.375} C_VEL
LIN {X 0,Y 150.567,Z 432.351,A -85,B 0,C 180,E1 -23948.272,E2 -23948.272} C_VEL
LIN {X 0,Y 149.218,Z 420.409,A -85,B 0,C 180,E1 -23950.083,E2 -23950.083} C_VEL
LIN {X 0,Y 149.062,Z 410.716,A -85,B 0,C 180,E1 -23960.709,E2 -23960.709} C_VEL
LIN {X 0,Y 149.564,Z 406.839,A -85,B 0,C 180,E1 -23965.019,E2 -23965.019} C_VEL
LIN {X 0,Y 150.503,Z 401.739,A -85,B 0,C 180,E1 -23970.909,E2 -23970.909} C_VEL
LIN {X 0,Y 150.422,Z 401.735,A -85,B 0,C 180,E1 -23974.102,E2 -23974.102} C_VEL
LIN {X 0,Y 150.276,Z 401.765,A -85,B 0,C 180,E1 -23977.444,E2 -23977.444} C_VEL
LIN {X 0,Y 150.159,Z 401.776,A -85,B 0,C 180,E1 -23981.508,E2 -23981.508} C_VEL
LIN {X 0,Y 150.128,Z 401.783,A -85,B 0,C 180,E1 -23985.396,E2 -23985.396} C_VEL
LIN {X 0,Y 150.153,Z 401.779,A -85,B 0,C 180,E1 -23989.059,E2 -23989.059} C_VEL
LIN {X 0,Y 150.181,Z 401.774,A -85,B 0,C 180,E1 -23992.708,E2 -23992.708} C_VEL
LIN {X 0,Y 150.217,Z 401.771,A -85,B 0,C 180,E1 -23997.368,E2 -23997.368} C_VEL
LIN {X 0,Y 150.247,Z 401.77,A -85,B 0,C 180,E1 -24002.718,E2 -24002.718} C_VEL
LIN {X 0,Y 150.355,Z 401.751,A -85,B 0,C 180,E1 -24009.206,E2 -24009.206} C_VEL
LIN {X 0,Y 150.373,Z 401.753,A -85,B 0,C 180,E1 -24013.714,E2 -24013.714} C_VEL
LIN {X 0,Y 150.614,Z 401.721,A -85,B 0,C 180,E1 -24019.242,E2 -24019.242} C_VEL
LIN {X 0,Y 150.708,Z 401.713,A -85,B 0,C 180,E1 -24021.958,E2 -24021.958} C_VEL
LIN {X 0,Y 151.221,Z 401.65,A -85,B 0,C 180,E1 -24030,E2 -24030} C_VEL
LIN {X 0,Y 150.747,Z 401.708,A -85,B 0,C 180,E1 -24038.04,E2 -24038.04} C_VEL
LIN {X 0,Y 150.617,Z 401.721,A -85,B 0,C 180,E1 -24041.507,E2 -24041.507} C_VEL
LIN {X 0,Y 150.399,Z 401.75,A -85,B 0,C 180,E1 -24046.282,E2 -24046.282} C_VEL
LIN {X 0,Y 150.392,Z 401.746,A -85,B 0,C 180,E1 -24050.831,E2 -24050.831} C_VEL
LIN {X 0,Y 150.247,Z 401.77,A -85,B 0,C 180,E1 -24057.282,E2 -24057.282} C_VEL
LIN {X 0,Y 150.22,Z 401.771,A -85,B 0,C 180,E1 -24062.634,E2 -24062.634} C_VEL
LIN {X 0,Y 150.213,Z 401.769,A -85,B 0,C 180,E1 -24067.462,E2 -24067.462} C_VEL
LIN {X 0,Y 150.155,Z 401.782,A -85,B 0,C 180,E1 -24071.506,E2 -24071.506} C_VEL
LIN {X 0,Y 150.127,Z 401.782,A -85,B 0,C 180,E1 -24075.395,E2 -24075.395} C_VEL
LIN {X 0,Y 150.142,Z 401.78,A -85,B 0,C 180,E1 -24079.055,E2 -24079.055} C_VEL
LIN {X 0,Y 150.183,Z 401.777,A -85,B 0,C 180,E1 -24082.706,E2 -24082.706} C_VEL
LIN {X 0,Y 150.221,Z 401.771,A -85,B 0,C 180,E1 -24087.364,E2 -24087.364} C_VEL
LIN {X 0,Y 150.247,Z 401.767,A -85,B 0,C 180,E1 -24092.717,E2 -24092.717} C_VEL
LIN {X 0,Y 150.354,Z 401.756,A -85,B 0,C 180,E1 -24099.206,E2 -24099.206} C_VEL
LIN {X 0,Y 150.392,Z 401.746,A -85,B 0,C 180,E1 -24103.716,E2 -24103.716} C_VEL
LIN {X 0,Y 150.691,Z 401.712,A -85,B 0,C 180,E1 -24109.248,E2 -24109.248} C_VEL
LIN {X 0,Y 150.765,Z 401.699,A -85,B 0,C 180,E1 -24111.961,E2 -24111.961} C_VEL
LIN {X 0,Y 151.22,Z 401.643,A -85,B 0,C 180,E1 -24120,E2 -24120} C_VEL
LIN {X 0,Y 150.765,Z 401.701,A -85,B 0,C 180,E1 -24128.039,E2 -24128.039} C_VEL
LIN {X 0,Y 150.636,Z 401.719,A -85,B 0,C 180,E1 -24131.546,E2 -24131.546} C_VEL
LIN {X 0,Y 150.384,Z 401.747,A -85,B 0,C 180,E1 -24136.284,E2 -24136.284} C_VEL
LIN {X 0,Y 150.352,Z 401.756,A -85,B 0,C 180,E1 -24140.793,E2 -24140.793} C_VEL
LIN {X 0,Y 150.245,Z 401.766,A -85,B 0,C 180,E1 -24147.282,E2 -24147.282} C_VEL
LIN {X 0,Y 150.218,Z 401.769,A -85,B 0,C 180,E1 -24152.634,E2 -24152.634} C_VEL
LIN {X 0,Y 150.212,Z 401.773,A -85,B 0,C 180,E1 -24157.462,E2 -24157.462} C_VEL
LIN {X 0,Y 150.38,Z 401.771,A -85,B 0,C 180,E1 -24164.781,E2 -24164.781} C_VEL
LIN {X 0,Y 151.786,Z 408.015,A -85,B 0,C 180,E1 -24170.512,E2 -24170.512} C_VEL
LIN {X 0,Y 153.595,Z 415.004,A -85,B 0,C 180,E1 -24176.696,E2 -24176.696} C_VEL
LIN {X 0,Y 153.703,Z 416.854,A -85,B 0,C 180,E1 -24178.276,E2 -24178.276} C_VEL
LIN {X 0,Y 151.016,Z 424.784,A -85,B 0,C 180,E1 -24185.238,E2 -24185.238} C_VEL
LIN {X 0,Y 150.279,Z 432.977,A -85,B 0,C 180,E1 -24192.655,E2 -24192.655} C_VEL
LIN {X 0,Y 150.338,Z 433.184,A -85,B 0,C 180,E1 -24192.837,E2 -24192.837} C_VEL
LIN {X 0,Y 150.759,Z 445.898,A -85,B 0,C 180,E1 -24194.453,E2 -24194.453} C_VEL
LIN {X 0,Y 151.924,Z 458.779,A -85,B 0,C 180,E1 -24196.627,E2 -24196.627} C_VEL
LIN {X 0,Y 152.824,Z 467.106,A -85,B 0,C 180,E1 -24198.393,E2 -24198.393} C_VEL
LIN {X 0,Y 152.602,Z 477.612,A -85,B 0,C 180,E1 -24201.392,E2 -24201.392} C_VEL
LIN {X 0,Y 152.681,Z 486.907,A -85,B 0,C 180,E1 -24204.718,E2 -24204.718} C_VEL
LIN {X 0,Y 153.118,Z 494.416,A -85,B 0,C 180,E1 -24208.027,E2 -24208.027} C_VEL
LIN {X 0,Y 153.104,Z 499.105,A -85,B 0,C 180,E1 -24210.658,E2 -24210.658} C_VEL
LIN {X 0,Y 152.85,Z 501.921,A -85,B 0,C 180,E1 -24212.636,E2 -24212.636} C_VEL
LIN {X 0,Y 151.49,Z 506.144,A -85,B 0,C 180,E1 -24216.66,E2 -24216.66} C_VEL
LIN {X 0,Y 150.774,Z 510.152,A -85,B 0,C 180,E1 -24221.8,E2 -24221.8} C_VEL
LIN {X 0,Y 151.313,Z 512.612,A -85,B 0,C 180,E1 -24226.182,E2 -24226.182} C_VEL
LIN {X 0,Y 153.602,Z 514.646,A -85,B 0,C 180,E1 -24231.472,E2 -24231.472} C_VEL
LIN {X 0,Y 157.526,Z 515.56,A -85,B 0,C 180,E1 -24236.497,E2 -24236.497} C_VEL
LIN {X 0,Y 163.122,Z 515.39,A -85,B 0,C 180,E1 -24241.132,E2 -24241.132} C_VEL
LIN {X 0,Y 170.205,Z 514.136,A -85,B 0,C 180,E1 -24245.316,E2 -24245.316} C_VEL
LIN {X 0,Y 178.457,Z 511.73,A -85,B 0,C 180,E1 -24249.059,E2 -24249.059} C_VEL
LIN {X 0,Y 187.891,Z 508.071,A -85,B 0,C 180,E1 -24252.321,E2 -24252.321} C_VEL
LIN {X 0,Y 192.603,Z 505.819,A -85,B 0,C 180,E1 -24253.893,E2 -24253.893} C_VEL
LIN {X 0,Y 194.163,Z 503.964,A -85,B 0,C 180,E1 -24256.549,E2 -24256.549} C_VEL
LIN {X 0,Y 193.188,Z 502.999,A -85,B 0,C 180,E1 -24259.815,E2 -24259.815} C_VEL
LIN {X 0,Y 192.216,Z 502.786,A -85,B 0,C 180,E1 -24261.569,E2 -24261.569} C_VEL
LIN {X 0,Y 189.285,Z 502.899,A -85,B 0,C 180,E1 -24264.77,E2 -24264.77} C_VEL
LIN {X 0,Y 188.233,Z 502.978,A -85,B 0,C 180,E1 -24265.61,E2 -24265.61} C_VEL
LIN {X 0,Y 186.436,Z 503.261,A -85,B 0,C 180,E1 -24266.415,E2 -24266.415} C_VEL
LIN {X 0,Y 182.612,Z 503.893,A -85,B 0,C 180,E1 -24267.203,E2 -24267.203} C_VEL
LIN {X 0,Y 173.687,Z 504.783,A -85,B 0,C 180,E1 -24268.45,E2 -24268.45} C_VEL
LIN {X 0,Y 170.513,Z 504.642,A -85,B 0,C 180,E1 -24269.335,E2 -24269.335} C_VEL
LIN {X 0,Y 164.72,Z 503.654,A -85,B 0,C 180,E1 -24272.009,E2 -24272.009} C_VEL
LIN {X 0,Y 160.84,Z 502.366,A -85,B 0,C 180,E1 -24274.09,E2 -24274.09} C_VEL
LIN {X 0,Y 155.579,Z 499.621,A -85,B 0,C 180,E1 -24277.42,E2 -24277.42} C_VEL
LIN {X 0,Y 151.108,Z 495.844,A -85,B 0,C 180,E1 -24281,E2 -24281} C_VEL
LIN {X 0,Y 147.565,Z 490.925,A -85,B 0,C 180,E1 -24284.815,E2 -24284.815} C_VEL
LIN {X 0,Y 144.936,Z 484.86,A -85,B 0,C 180,E1 -24288.816,E2 -24288.816} C_VEL
LIN {X 0,Y 143.384,Z 477.344,A -85,B 0,C 180,E1 -24292.962,E2 -24292.962} C_VEL
LIN {X 0,Y 142.751,Z 468.24,A -85,B 0,C 180,E1 -24297.178,E2 -24297.178} C_VEL
LIN {X 0,Y 142.919,Z 457.803,A -85,B 0,C 180,E1 -24301.057,E2 -24301.057} C_VEL
LIN {X 0,Y 143.212,Z 448.467,A -85,B 0,C 180,E1 -24303.869,E2 -24303.869} C_VEL
LIN {X 0,Y 143.546,Z 436.918,A -85,B 0,C 180,E1 -24306.678,E2 -24306.678} C_VEL
LIN {X 0,Y 143.571,Z 431.618,A -85,B 0,C 180,E1 -24307.737,E2 -24307.737} C_VEL
LIN {X 0,Y 142.328,Z 420.747,A -85,B 0,C 180,E1 -24309.435,E2 -24309.435} C_VEL
LIN {X 0,Y 141.43,Z 416.384,A -85,B 0,C 180,E1 -24314.387,E2 -24314.387} C_VEL
LIN {X 0,Y 141.909,Z 411.276,A -85,B 0,C 180,E1 -24320.284,E2 -24320.284} C_VEL
LIN {X 0,Y 142.609,Z 406.079,A -85,B 0,C 180,E1 -24326.33,E2 -24326.33} C_VEL
LIN {X 0,Y 143.355,Z 402.629,A -85,B 0,C 180,E1 -24330.573,E2 -24330.573} C_VEL
LIN {X 0,Y 143.426,Z 402.605,A -85,B 0,C 180,E1 -24333.589,E2 -24333.589} C_VEL
LIN {X 0,Y 143.097,Z 402.659,A -85,B 0,C 180,E1 -24339.679,E2 -24339.679} C_VEL
LIN {X 0,Y 143.06,Z 402.66,A -85,B 0,C 180,E1 -24343.454,E2 -24343.454} C_VEL
LIN {X 0,Y 143.067,Z 402.663,A -85,B 0,C 180,E1 -24347.465,E2 -24347.465} C_VEL
LIN {X 0,Y 143.079,Z 402.655,A -85,B 0,C 180,E1 -24351.806,E2 -24351.806} C_VEL
LIN {X 0,Y 143.184,Z 402.647,A -85,B 0,C 180,E1 -24357.321,E2 -24357.321} C_VEL
LIN {X 0,Y 143.193,Z 402.645,A -85,B 0,C 180,E1 -24362.063,E2 -24362.063} C_VEL
LIN {X 0,Y 143.28,Z 402.632,A -85,B 0,C 180,E1 -24368.744,E2 -24368.744} C_VEL
LIN {X 0,Y 143.311,Z 402.633,A -85,B 0,C 180,E1 -24372.888,E2 -24372.888} C_VEL
LIN {X 0,Y 143.54,Z 402.603,A -85,B 0,C 180,E1 -24378.705,E2 -24378.705} C_VEL
LIN {X 0,Y 143.629,Z 402.593,A -85,B 0,C 180,E1 -24381.559,E2 -24381.559} C_VEL
LIN {X 0,Y 144.179,Z 402.527,A -85,B 0,C 180,E1 -24390,E2 -24390} C_VEL
LIN {X 0,Y 143.668,Z 402.589,A -85,B 0,C 180,E1 -24398.439,E2 -24398.439} C_VEL
LIN {X 0,Y 143.55,Z 402.599,A -85,B 0,C 180,E1 -24401.712,E2 -24401.712} C_VEL
LIN {X 0,Y 143.338,Z 402.63,A -85,B 0,C 180,E1 -24407.109,E2 -24407.109} C_VEL
LIN {X 0,Y 143.313,Z 402.628,A -85,B 0,C 180,E1 -24411.289,E2 -24411.289} C_VEL
LIN {X 0,Y 143.193,Z 402.645,A -85,B 0,C 180,E1 -24417.937,E2 -24417.937} C_VEL
LIN {X 0,Y 143.171,Z 402.651,A -85,B 0,C 180,E1 -24423.435,E2 -24423.435} C_VEL
LIN {X 0,Y 143.076,Z 402.659,A -85,B 0,C 180,E1 -24429.685,E2 -24429.685} C_VEL
LIN {X 0,Y 143.058,Z 402.665,A -85,B 0,C 180,E1 -24433.454,E2 -24433.454} C_VEL
LIN {X 0,Y 143.04,Z 402.662,A -85,B 0,C 180,E1 -24437.476,E2 -24437.476} C_VEL
LIN {X 0,Y 143.08,Z 402.662,A -85,B 0,C 180,E1 -24441.805,E2 -24441.805} C_VEL
LIN {X 0,Y 143.188,Z 402.647,A -85,B 0,C 180,E1 -24447.322,E2 -24447.322} C_VEL
LIN {X 0,Y 143.194,Z 402.646,A -85,B 0,C 180,E1 -24452.061,E2 -24452.061} C_VEL
LIN {X 0,Y 143.279,Z 402.638,A -85,B 0,C 180,E1 -24458.744,E2 -24458.744} C_VEL
LIN {X 0,Y 143.325,Z 402.626,A -85,B 0,C 180,E1 -24462.889,E2 -24462.889} C_VEL
LIN {X 0,Y 143.604,Z 402.596,A -85,B 0,C 180,E1 -24468.711,E2 -24468.711} C_VEL
LIN {X 0,Y 143.686,Z 402.58,A -85,B 0,C 180,E1 -24471.562,E2 -24471.562} C_VEL
LIN {X 0,Y 144.179,Z 402.519,A -85,B 0,C 180,E1 -24480,E2 -24480} C_VEL
LIN {X 0,Y 143.686,Z 402.581,A -85,B 0,C 180,E1 -24488.438,E2 -24488.438} C_VEL
LIN {X 0,Y 143.572,Z 402.6,A -85,B 0,C 180,E1 -24491.757,E2 -24491.757} C_VEL
LIN {X 0,Y 143.318,Z 402.625,A -85,B 0,C 180,E1 -24497.111,E2 -24497.111} C_VEL
LIN {X 0,Y 143.278,Z 402.637,A -85,B 0,C 180,E1 -24501.255,E2 -24501.255} C_VEL
LIN {X 0,Y 143.191,Z 402.647,A -85,B 0,C 180,E1 -24507.937,E2 -24507.937} C_VEL
LIN {X 0,Y 143.169,Z 402.647,A -85,B 0,C 180,E1 -24513.435,E2 -24513.435} C_VEL
LIN {X 0,Y 143.092,Z 402.662,A -85,B 0,C 180,E1 -24519.68,E2 -24519.68} C_VEL
LIN {X 0,Y 143.361,Z 402.796,A -85,B 0,C 180,E1 -24525.054,E2 -24525.054} C_VEL
LIN {X 0,Y 144.804,Z 408.915,A -85,B 0,C 180,E1 -24530.946,E2 -24530.946} C_VEL
LIN {X 0,Y 146.461,Z 415.014,A -85,B 0,C 180,E1 -24536.636,E2 -24536.636} C_VEL
LIN {X 0,Y 146.578,Z 416.71,A -85,B 0,C 180,E1 -24538.169,E2 -24538.169} C_VEL
LIN {X 0,Y 143.841,Z 424.529,A -85,B 0,C 180,E1 -24545.461,E2 -24545.461} C_VEL
LIN {X 0,Y 143.251,Z 432.238,A -85,B 0,C 180,E1 -24552.881,E2 -24552.881} C_VEL
LIN {X 0,Y 143.422,Z 432.851,A -85,B 0,C 180,E1 -24553.452,E2 -24553.452} C_VEL
LIN {X 0,Y 143.981,Z 446.439,A -85,B 0,C 180,E1 -24555.333,E2 -24555.333} C_VEL
LIN {X 0,Y 145.182,Z 458.272,A -85,B 0,C 180,E1 -24557.444,E2 -24557.444} C_VEL
LIN {X 0,Y 146.084,Z 465.022,A -85,B 0,C 180,E1 -24558.905,E2 -24558.905} C_VEL
LIN {X 0,Y 145.932,Z 474.733,A -85,B 0,C 180,E1 -24561.693,E2 -24561.693} C_VEL
LIN {X 0,Y 146.074,Z 484.424,A -85,B 0,C 180,E1 -24565.17,E2 -24565.17} C_VEL
LIN {X 0,Y 146.578,Z 492.095,A -85,B 0,C 180,E1 -24568.627,E2 -24568.627} C_VEL
LIN {X 0,Y 146.604,Z 496.872,A -85,B 0,C 180,E1 -24571.374,E2 -24571.374} C_VEL
LIN {X 0,Y 146.406,Z 498.837,A -85,B 0,C 180,E1 -24572.752,E2 -24572.752} C_VEL
LIN {X 0,Y 144.996,Z 503.41,A -85,B 0,C 180,E1 -24576.96,E2 -24576.96} C_VEL
LIN {X 0,Y 144.239,Z 508.103,A -85,B 0,C 180,E1 -24582.969,E2 -24582.969} C_VEL
LIN {X 0,Y 144.786,Z 510.428,A -85,B 0,C 180,E1 -24586.933,E2 -24586.933} C_VEL
LIN {X 0,Y 147.212,Z 512.804,A -85,B 0,C 180,E1 -24592.453,E2 -24592.453} C_VEL
LIN {X 0,Y 151.309,Z 514.074,A -85,B 0,C 180,E1 -24597.677,E2 -24597.677} C_VEL
LIN {X 0,Y 157.145,Z 514.339,A -85,B 0,C 180,E1 -24602.458,E2 -24602.458} C_VEL
LIN {X 0,Y 164.475,Z 513.549,A -85,B 0,C 180,E1 -24606.743,E2 -24606.743} C_VEL
LIN {X 0,Y 173.02,Z 511.649,A -85,B 0,C 180,E1 -24610.535,E2 -24610.535} C_VEL
LIN {X 0,Y 182.713,Z 508.556,A -85,B 0,C 180,E1 -24613.818,E2 -24613.818} C_VEL
LIN {X 0,Y 186.702,Z 506.705,A -85,B 0,C 180,E1 -24615.661,E2 -24615.661} C_VEL
LIN {X 0,Y 187.102,Z 505.82,A -85,B 0,C 180,E1 -24617.458,E2 -24617.458} C_VEL
LIN {X 0,Y 186.19,Z 505.094,A -85,B 0,C 180,E1 -24620.082,E2 -24620.082} C_VEL
LIN {X 0,Y 184.392,Z 504.781,A -85,B 0,C 180,E1 -24622.423,E2 -24622.423} C_VEL
LIN {X 0,Y 182.08,Z 504.675,A -85,B 0,C 180,E1 -24624.621,E2 -24624.621} C_VEL
LIN {X 0,Y 177.959,Z 504.896,A -85,B 0,C 180,E1 -24626.434,E2 -24626.434} C_VEL
LIN {X 0,Y 170.513,Z 504.642,A -85,B 0,C 180,E1 -24629.335,E2 -24629.335} C_VEL
LIN {X 0,Y 166.422,Z 504.232,A -85,B 0,C 180,E1 -24630.779,E2 -24630.779} C_VEL
LIN {X 0,Y 158.678,Z 502.816,A -85,B 0,C 180,E1 -24632.909,E2 -24632.909} C_VEL
LIN {X 0,Y 152.752,Z 500.97,A -85,B 0,C 180,E1 -24634.722,E2 -24634.722} C_VEL
LIN {X 0,Y 149.154,Z 499.17,A -85,B 0,C 180,E1 -24636.357,E2 -24636.357} C_VEL
LIN {X 0,Y 148.231,Z 498.488,A -85,B 0,C 180,E1 -24636.975,E2 -24636.975} C_VEL
LIN {X 0,Y 143.15,Z 493.307,A -85,B 0,C 180,E1 -24641.39,E2 -24641.39} C_VEL
LIN {X 0,Y 139.338,Z 486.474,A -85,B 0,C 180,E1 -24646.138,E2 -24646.138} C_VEL
LIN {X 0,Y 136.992,Z 477.961,A -85,B 0,C 180,E1 -24651.147,E2 -24651.147} C_VEL
LIN {X 0,Y 136.127,Z 468.817,A -85,B 0,C 180,E1 -24655.559,E2 -24655.559} C_VEL
LIN {X 0,Y 136.051,Z 458.625,A -85,B 0,C 180,E1 -24659.63,E2 -24659.63} C_VEL
LIN {X 0,Y 136.38,Z 449.503,A -85,B 0,C 180,E1 -24662.585,E2 -24662.585} C_VEL
LIN {X 0,Y 136.666,Z 438.116,A -85,B 0,C 180,E1 -24665.533,E2 -24665.533} C_VEL
LIN {X 0,Y 136.704,Z 431.083,A -85,B 0,C 180,E1 -24667.014,E2 -24667.014} C_VEL
LIN {X 0,Y 135.464,Z 421.089,A -85,B 0,C 180,E1 -24668.672,E2 -24668.672} C_VEL
LIN {X 0,Y 134.361,Z 415.645,A -85,B 0,C 180,E1 -24675.161,E2 -24675.161} C_VEL
